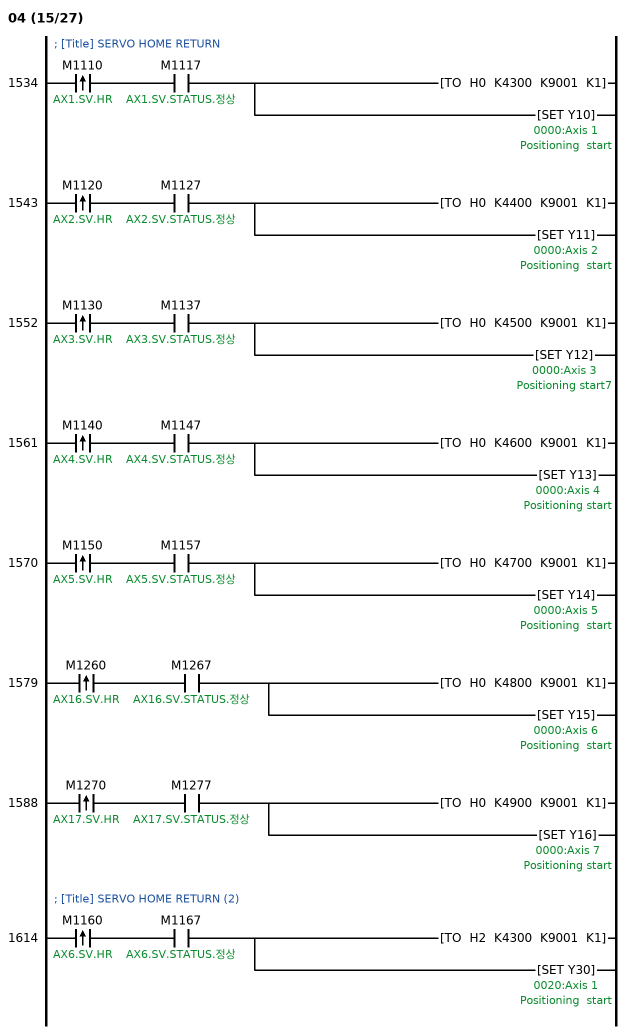
; [Title] SERVO HOME RETURN
1534  LDP     M1110  ; AX1.SV.HR
      AND     M1117  ; AX1.SV.STATUS.정상
      TO      H0 K4300 K9001 K1
      SET     Y10  ; 0000:Axis 1  Positioning  start
1543  LDP     M1120  ; AX2.SV.HR
      AND     M1127  ; AX2.SV.STATUS.정상
      TO      H0 K4400 K9001 K1
      SET     Y11  ; 0000:Axis 2  Positioning  start
1552  LDP     M1130  ; AX3.SV.HR
      AND     M1137  ; AX3.SV.STATUS.정상
      TO      H0 K4500 K9001 K1
      SET     Y12  ; 0000:Axis 3 Positioning start7
1561  LDP     M1140  ; AX4.SV.HR
      AND     M1147  ; AX4.SV.STATUS.정상
      TO      H0 K4600 K9001 K1
      SET     Y13  ; 0000:Axis 4 Positioning start
1570  LDP     M1150  ; AX5.SV.HR
      AND     M1157  ; AX5.SV.STATUS.정상
      TO      H0 K4700 K9001 K1
      SET     Y14  ; 0000:Axis 5  Positioning  start
1579  LDP     M1260  ; AX16.SV.HR
      AND     M1267  ; AX16.SV.STATUS.정상
      TO      H0 K4800 K9001 K1
      SET     Y15  ; 0000:Axis 6  Positioning  start
1588  LDP     M1270  ; AX17.SV.HR
      AND     M1277  ; AX17.SV.STATUS.정상
      TO      H0 K4900 K9001 K1
      SET     Y16  ; 0000:Axis 7 Positioning start
; [Title] SERVO HOME RETURN (2)
1614  LDP     M1160  ; AX6.SV.HR
      AND     M1167  ; AX6.SV.STATUS.정상
      TO      H2 K4300 K9001 K1
      SET     Y30  ; 0020:Axis 1  Positioning  start
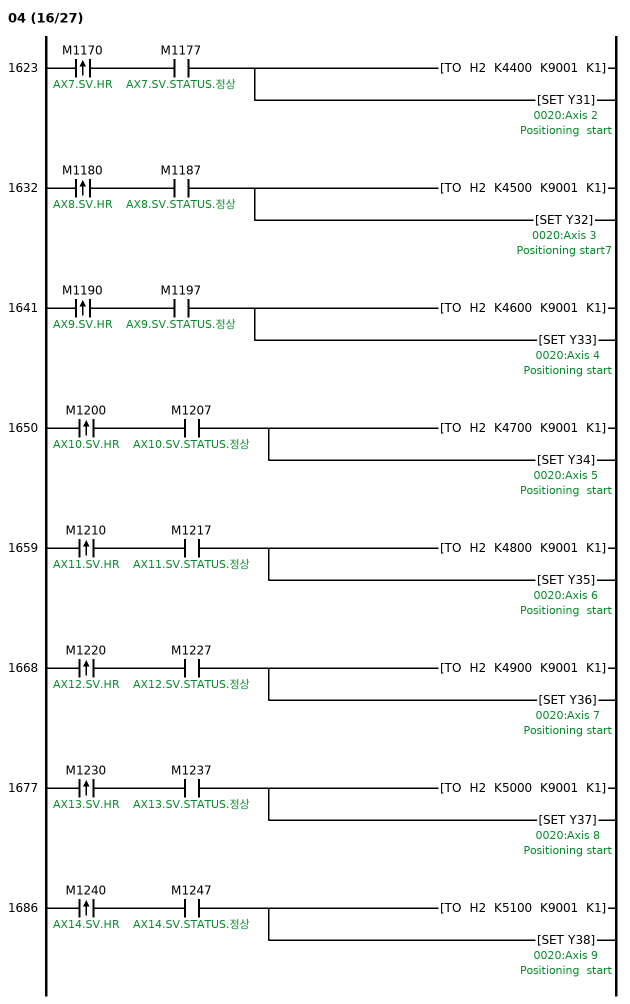
1623  LDP     M1170  ; AX7.SV.HR
      AND     M1177  ; AX7.SV.STATUS.정상
      TO      H2 K4400 K9001 K1
      SET     Y31  ; 0020:Axis 2  Positioning  start
1632  LDP     M1180  ; AX8.SV.HR
      AND     M1187  ; AX8.SV.STATUS.정상
      TO      H2 K4500 K9001 K1
      SET     Y32  ; 0020:Axis 3 Positioning start7
1641  LDP     M1190  ; AX9.SV.HR
      AND     M1197  ; AX9.SV.STATUS.정상
      TO      H2 K4600 K9001 K1
      SET     Y33  ; 0020:Axis 4 Positioning start
1650  LDP     M1200  ; AX10.SV.HR
      AND     M1207  ; AX10.SV.STATUS.정상
      TO      H2 K4700 K9001 K1
      SET     Y34  ; 0020:Axis 5  Positioning  start
1659  LDP     M1210  ; AX11.SV.HR
      AND     M1217  ; AX11.SV.STATUS.정상
      TO      H2 K4800 K9001 K1
      SET     Y35  ; 0020:Axis 6  Positioning  start
1668  LDP     M1220  ; AX12.SV.HR
      AND     M1227  ; AX12.SV.STATUS.정상
      TO      H2 K4900 K9001 K1
      SET     Y36  ; 0020:Axis 7 Positioning start
1677  LDP     M1230  ; AX13.SV.HR
      AND     M1237  ; AX13.SV.STATUS.정상
      TO      H2 K5000 K9001 K1
      SET     Y37  ; 0020:Axis 8 Positioning start
1686  LDP     M1240  ; AX14.SV.HR
      AND     M1247  ; AX14.SV.STATUS.정상
      TO      H2 K5100 K9001 K1
      SET     Y38  ; 0020:Axis 9  Positioning  start
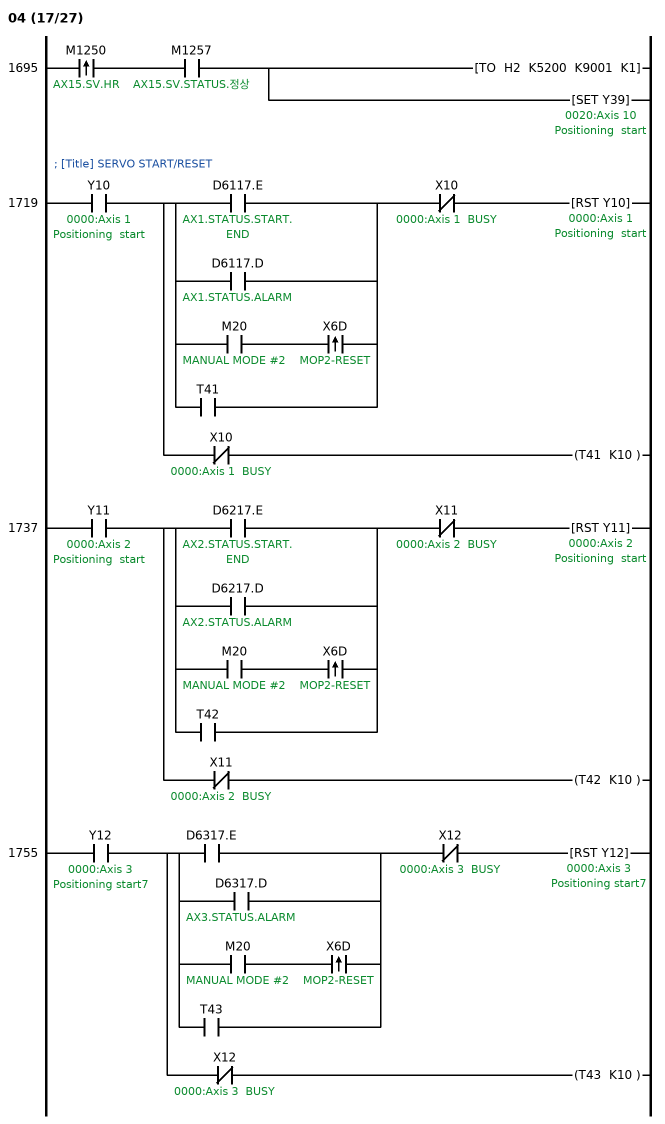
1695  LDP     M1250  ; AX15.SV.HR
      AND     M1257  ; AX15.SV.STATUS.정상
      TO      H2 K5200 K9001 K1
      SET     Y39  ; 0020:Axis 10  Positioning  start
; [Title] SERVO START/RESET
1719  LD      Y10  ; 0000:Axis 1  Positioning  start
      MPS
      LD      D6117.E  ; AX1.STATUS.START.END
      OR      D6117.D  ; AX1.STATUS.ALARM
      LD      M20  ; MANUAL MODE #2
      ANDP    X6D  ; MOP2-RESET
      ORB
      OR      T41
      ANB
      ANI     X10  ; 0000:Axis 1  BUSY
      RST     Y10  ; 0000:Axis 1  Positioning  start
      MPP
      ANI     X10  ; 0000:Axis 1  BUSY
      OUT     T41 K10
1737  LD      Y11  ; 0000:Axis 2  Positioning  start
      MPS
      LD      D6217.E  ; AX2.STATUS.START.END
      OR      D6217.D  ; AX2.STATUS.ALARM
      LD      M20  ; MANUAL MODE #2
      ANDP    X6D  ; MOP2-RESET
      ORB
      OR      T42
      ANB
      ANI     X11  ; 0000:Axis 2  BUSY
      RST     Y11  ; 0000:Axis 2  Positioning  start
      MPP
      ANI     X11  ; 0000:Axis 2  BUSY
      OUT     T42 K10
1755  LD      Y12  ; 0000:Axis 3 Positioning start7
      MPS
      LD      D6317.E
      OR      D6317.D  ; AX3.STATUS.ALARM
      LD      M20  ; MANUAL MODE #2
      ANDP    X6D  ; MOP2-RESET
      ORB
      OR      T43
      ANB
      ANI     X12  ; 0000:Axis 3  BUSY
      RST     Y12  ; 0000:Axis 3 Positioning start7
      MPP
      ANI     X12  ; 0000:Axis 3  BUSY
      OUT     T43 K10
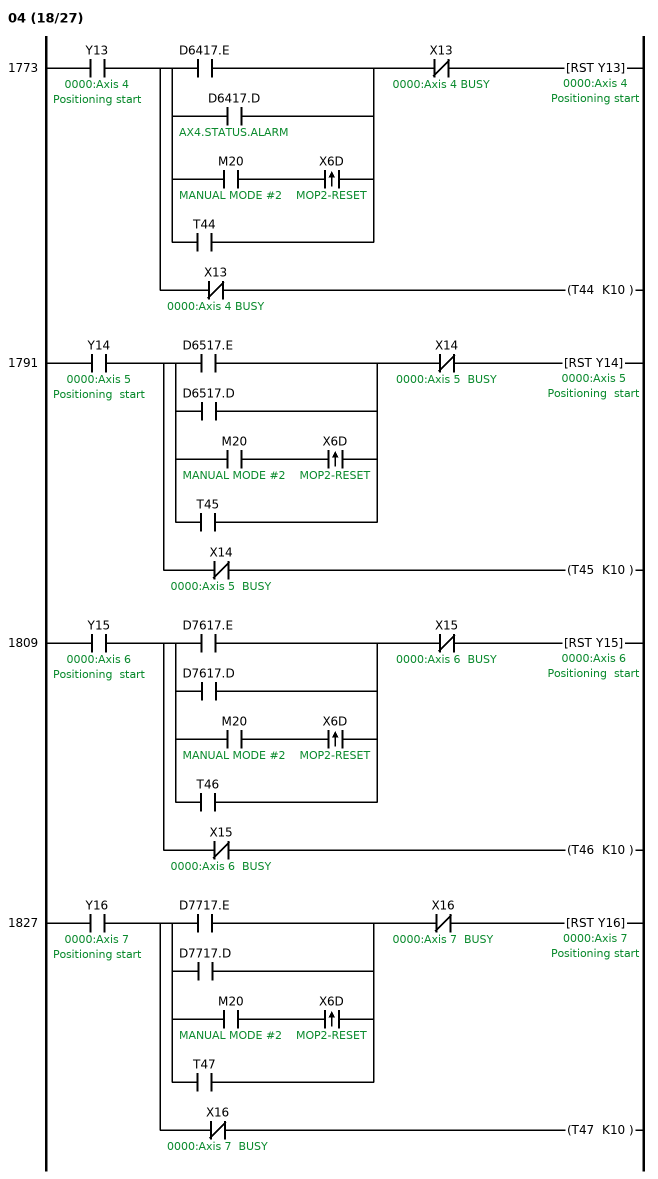
1773  LD      Y13  ; 0000:Axis 4 Positioning start
      MPS
      LD      D6417.E
      OR      D6417.D  ; AX4.STATUS.ALARM
      LD      M20  ; MANUAL MODE #2
      ANDP    X6D  ; MOP2-RESET
      ORB
      OR      T44
      ANB
      ANI     X13  ; 0000:Axis 4 BUSY
      RST     Y13  ; 0000:Axis 4 Positioning start
      MPP
      ANI     X13  ; 0000:Axis 4 BUSY
      OUT     T44 K10
1791  LD      Y14  ; 0000:Axis 5  Positioning  start
      MPS
      LD      D6517.E
      OR      D6517.D
      LD      M20  ; MANUAL MODE #2
      ANDP    X6D  ; MOP2-RESET
      ORB
      OR      T45
      ANB
      ANI     X14  ; 0000:Axis 5  BUSY
      RST     Y14  ; 0000:Axis 5  Positioning  start
      MPP
      ANI     X14  ; 0000:Axis 5  BUSY
      OUT     T45 K10
1809  LD      Y15  ; 0000:Axis 6  Positioning  start
      MPS
      LD      D7617.E
      OR      D7617.D
      LD      M20  ; MANUAL MODE #2
      ANDP    X6D  ; MOP2-RESET
      ORB
      OR      T46
      ANB
      ANI     X15  ; 0000:Axis 6  BUSY
      RST     Y15  ; 0000:Axis 6  Positioning  start
      MPP
      ANI     X15  ; 0000:Axis 6  BUSY
      OUT     T46 K10
1827  LD      Y16  ; 0000:Axis 7 Positioning start
      MPS
      LD      D7717.E
      OR      D7717.D
      LD      M20  ; MANUAL MODE #2
      ANDP    X6D  ; MOP2-RESET
      ORB
      OR      T47
      ANB
      ANI     X16  ; 0000:Axis 7  BUSY
      RST     Y16  ; 0000:Axis 7 Positioning start
      MPP
      ANI     X16  ; 0000:Axis 7  BUSY
      OUT     T47 K10
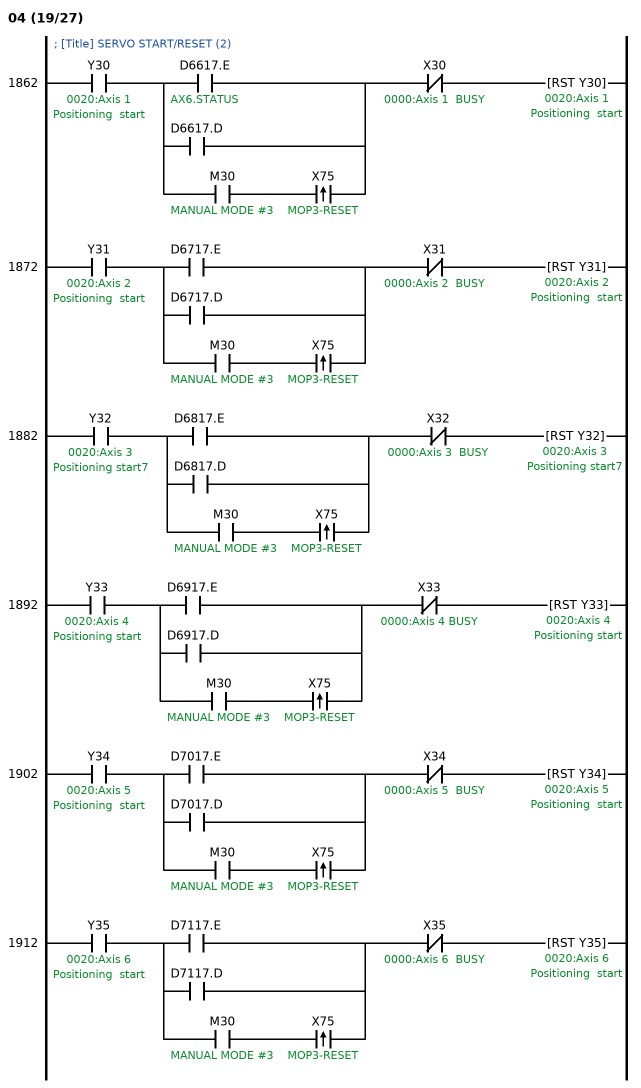
; [Title] SERVO START/RESET (2)
1862  LD      Y30  ; 0020:Axis 1  Positioning  start
      LD      D6617.E  ; AX6.STATUS
      OR      D6617.D
      LD      M30  ; MANUAL MODE #3
      ANDP    X75  ; MOP3-RESET
      ORB
      ANB
      ANI     X30  ; 0000:Axis 1  BUSY
      RST     Y30  ; 0020:Axis 1  Positioning  start
1872  LD      Y31  ; 0020:Axis 2  Positioning  start
      LD      D6717.E
      OR      D6717.D
      LD      M30  ; MANUAL MODE #3
      ANDP    X75  ; MOP3-RESET
      ORB
      ANB
      ANI     X31  ; 0000:Axis 2  BUSY
      RST     Y31  ; 0020:Axis 2  Positioning  start
1882  LD      Y32  ; 0020:Axis 3 Positioning start7
      LD      D6817.E
      OR      D6817.D
      LD      M30  ; MANUAL MODE #3
      ANDP    X75  ; MOP3-RESET
      ORB
      ANB
      ANI     X32  ; 0000:Axis 3  BUSY
      RST     Y32  ; 0020:Axis 3 Positioning start7
1892  LD      Y33  ; 0020:Axis 4 Positioning start
      LD      D6917.E
      OR      D6917.D
      LD      M30  ; MANUAL MODE #3
      ANDP    X75  ; MOP3-RESET
      ORB
      ANB
      ANI     X33  ; 0000:Axis 4 BUSY
      RST     Y33  ; 0020:Axis 4 Positioning start
1902  LD      Y34  ; 0020:Axis 5  Positioning  start
      LD      D7017.E
      OR      D7017.D
      LD      M30  ; MANUAL MODE #3
      ANDP    X75  ; MOP3-RESET
      ORB
      ANB
      ANI     X34  ; 0000:Axis 5  BUSY
      RST     Y34  ; 0020:Axis 5  Positioning  start
1912  LD      Y35  ; 0020:Axis 6  Positioning  start
      LD      D7117.E
      OR      D7117.D
      LD      M30  ; MANUAL MODE #3
      ANDP    X75  ; MOP3-RESET
      ORB
      ANB
      ANI     X35  ; 0000:Axis 6  BUSY
      RST     Y35  ; 0020:Axis 6  Positioning  start
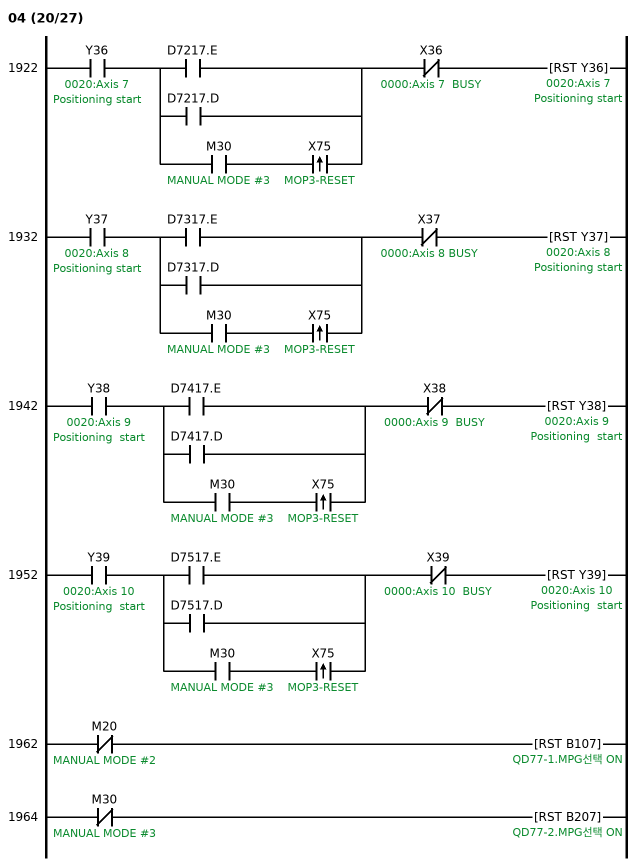
1922  LD      Y36  ; 0020:Axis 7 Positioning start
      LD      D7217.E
      OR      D7217.D
      LD      M30  ; MANUAL MODE #3
      ANDP    X75  ; MOP3-RESET
      ORB
      ANB
      ANI     X36  ; 0000:Axis 7  BUSY
      RST     Y36  ; 0020:Axis 7 Positioning start
1932  LD      Y37  ; 0020:Axis 8 Positioning start
      LD      D7317.E
      OR      D7317.D
      LD      M30  ; MANUAL MODE #3
      ANDP    X75  ; MOP3-RESET
      ORB
      ANB
      ANI     X37  ; 0000:Axis 8 BUSY
      RST     Y37  ; 0020:Axis 8 Positioning start
1942  LD      Y38  ; 0020:Axis 9  Positioning  start
      LD      D7417.E
      OR      D7417.D
      LD      M30  ; MANUAL MODE #3
      ANDP    X75  ; MOP3-RESET
      ORB
      ANB
      ANI     X38  ; 0000:Axis 9  BUSY
      RST     Y38  ; 0020:Axis 9  Positioning  start
1952  LD      Y39  ; 0020:Axis 10  Positioning  start
      LD      D7517.E
      OR      D7517.D
      LD      M30  ; MANUAL MODE #3
      ANDP    X75  ; MOP3-RESET
      ORB
      ANB
      ANI     X39  ; 0000:Axis 10  BUSY
      RST     Y39  ; 0020:Axis 10  Positioning  start
1962  LDI     M20  ; MANUAL MODE #2
      RST     B107  ; QD77-1.MPG선택 ON
1964  LDI     M30  ; MANUAL MODE #3
      RST     B207  ; QD77-2.MPG선택 ON
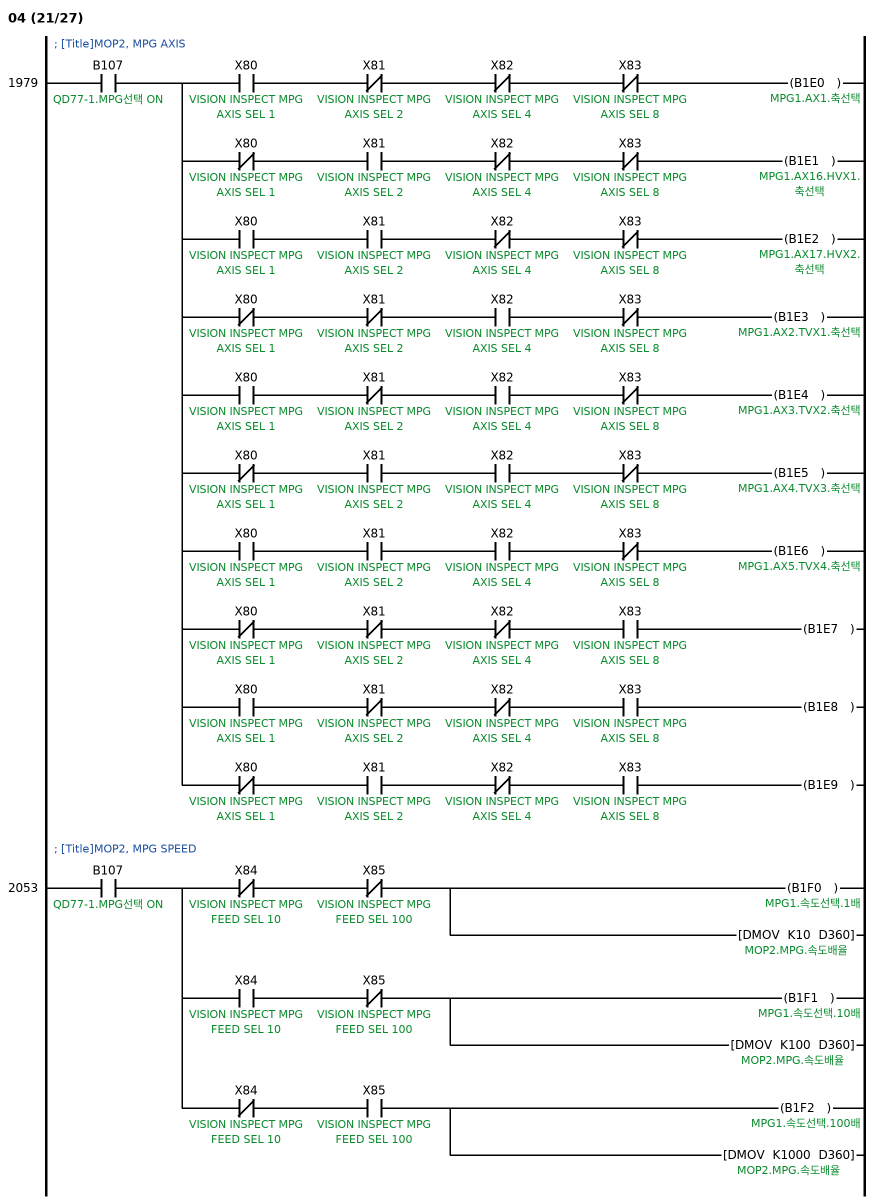
; [Title]MOP2, MPG AXIS
1979  LD      B107  ; QD77-1.MPG선택 ON
      MPS
      AND     X80  ; VISION INSPECT MPG AXIS SEL 1
      ANI     X81  ; VISION INSPECT MPG AXIS SEL 2
      ANI     X82  ; VISION INSPECT MPG AXIS SEL 4
      ANI     X83  ; VISION INSPECT MPG AXIS SEL 8
      OUT     B1E0  ; MPG1.AX1.축선택
      MRD
      ANI     X80  ; VISION INSPECT MPG AXIS SEL 1
      AND     X81  ; VISION INSPECT MPG AXIS SEL 2
      ANI     X82  ; VISION INSPECT MPG AXIS SEL 4
      ANI     X83  ; VISION INSPECT MPG AXIS SEL 8
      OUT     B1E1  ; MPG1.AX16.HVX1.축선택
      MRD
      AND     X80  ; VISION INSPECT MPG AXIS SEL 1
      AND     X81  ; VISION INSPECT MPG AXIS SEL 2
      ANI     X82  ; VISION INSPECT MPG AXIS SEL 4
      ANI     X83  ; VISION INSPECT MPG AXIS SEL 8
      OUT     B1E2  ; MPG1.AX17.HVX2.축선택
      MRD
      ANI     X80  ; VISION INSPECT MPG AXIS SEL 1
      ANI     X81  ; VISION INSPECT MPG AXIS SEL 2
      AND     X82  ; VISION INSPECT MPG AXIS SEL 4
      ANI     X83  ; VISION INSPECT MPG AXIS SEL 8
      OUT     B1E3  ; MPG1.AX2.TVX1.축선택
      MRD
      AND     X80  ; VISION INSPECT MPG AXIS SEL 1
      ANI     X81  ; VISION INSPECT MPG AXIS SEL 2
      AND     X82  ; VISION INSPECT MPG AXIS SEL 4
      ANI     X83  ; VISION INSPECT MPG AXIS SEL 8
      OUT     B1E4  ; MPG1.AX3.TVX2.축선택
      MRD
      ANI     X80  ; VISION INSPECT MPG AXIS SEL 1
      AND     X81  ; VISION INSPECT MPG AXIS SEL 2
      AND     X82  ; VISION INSPECT MPG AXIS SEL 4
      ANI     X83  ; VISION INSPECT MPG AXIS SEL 8
      OUT     B1E5  ; MPG1.AX4.TVX3.축선택
      MRD
      AND     X80  ; VISION INSPECT MPG AXIS SEL 1
      AND     X81  ; VISION INSPECT MPG AXIS SEL 2
      AND     X82  ; VISION INSPECT MPG AXIS SEL 4
      ANI     X83  ; VISION INSPECT MPG AXIS SEL 8
      OUT     B1E6  ; MPG1.AX5.TVX4.축선택
      MRD
      ANI     X80  ; VISION INSPECT MPG AXIS SEL 1
      ANI     X81  ; VISION INSPECT MPG AXIS SEL 2
      ANI     X82  ; VISION INSPECT MPG AXIS SEL 4
      AND     X83  ; VISION INSPECT MPG AXIS SEL 8
      OUT     B1E7
      MRD
      AND     X80  ; VISION INSPECT MPG AXIS SEL 1
      ANI     X81  ; VISION INSPECT MPG AXIS SEL 2
      ANI     X82  ; VISION INSPECT MPG AXIS SEL 4
      AND     X83  ; VISION INSPECT MPG AXIS SEL 8
      OUT     B1E8
      MPP
      ANI     X80  ; VISION INSPECT MPG AXIS SEL 1
      AND     X81  ; VISION INSPECT MPG AXIS SEL 2
      ANI     X82  ; VISION INSPECT MPG AXIS SEL 4
      AND     X83  ; VISION INSPECT MPG AXIS SEL 8
      OUT     B1E9
; [Title]MOP2, MPG SPEED
2053  LD      B107  ; QD77-1.MPG선택 ON
      MPS
      ANI     X84  ; VISION INSPECT MPG FEED SEL 10
      ANI     X85  ; VISION INSPECT MPG FEED SEL 100
      OUT     B1F0  ; MPG1.속도선택.1배
      DMOV    K10 D360  ; MOP2.MPG.속도배율
      MRD
      AND     X84  ; VISION INSPECT MPG FEED SEL 10
      ANI     X85  ; VISION INSPECT MPG FEED SEL 100
      OUT     B1F1  ; MPG1.속도선택.10배
      DMOV    K100 D360
      MPP
      ANI     X84  ; VISION INSPECT MPG FEED SEL 10
      AND     X85  ; VISION INSPECT MPG FEED SEL 100
      OUT     B1F2  ; MPG1.속도선택.100배
      DMOV    K1000 D360
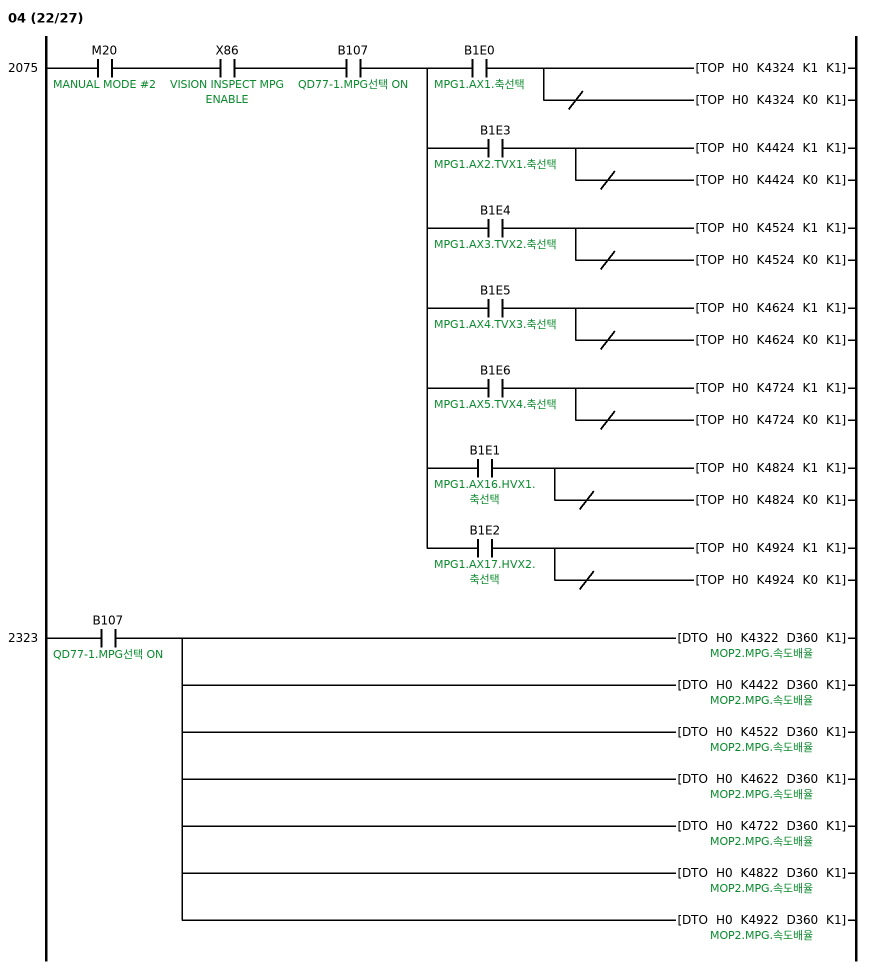
2075  LD      M20  ; MANUAL MODE #2
      AND     X86  ; VISION INSPECT MPG ENABLE
      AND     B107  ; QD77-1.MPG선택 ON
      MPS
      AND     B1E0  ; MPG1.AX1.축선택
      TOP     H0 K4324 K1 K1
        [note] MPG #1 AXIS 허가
      INV
      TOP     H0 K4324 K0 K1
        [note] MPG #1 AXIS 불가
      MRD
      AND     B1E3  ; MPG1.AX2.TVX1.축선택
      TOP     H0 K4424 K1 K1
        [note] MPG #2 AXIS 허가
      INV
      TOP     H0 K4424 K0 K1
        [note] MPG #2 AXIS 불가
      MRD
      AND     B1E4  ; MPG1.AX3.TVX2.축선택
      TOP     H0 K4524 K1 K1
        [note] MPG #3 AXIS 허가
      INV
      TOP     H0 K4524 K0 K1
        [note] MPG #3 AXIS 불가
      MRD
      AND     B1E5  ; MPG1.AX4.TVX3.축선택
      TOP     H0 K4624 K1 K1
        [note] MPG #4 AXIS 허가
      INV
      TOP     H0 K4624 K0 K1
        [note] MPG #4 AXIS 불가
      MRD
      AND     B1E6  ; MPG1.AX5.TVX4.축선택
      TOP     H0 K4724 K1 K1
        [note] MPG #5 AXIS 허가
      INV
      TOP     H0 K4724 K0 K1
        [note] MPG #5 AXIS 불가
      MRD
      AND     B1E1  ; MPG1.AX16.HVX1.축선택
      TOP     H0 K4824 K1 K1
        [note] MPG #6 AXIS 허가
      INV
      TOP     H0 K4824 K0 K1
        [note] MPG #6 AXIS 불가
      MPP
      AND     B1E2  ; MPG1.AX17.HVX2.축선택
      TOP     H0 K4924 K1 K1
        [note] MPG #7 AXIS 허가
      INV
      TOP     H0 K4924 K0 K1
        [note] MPG #7 AXIS 불가
2323  LD      B107  ; QD77-1.MPG선택 ON
      DTO     H0 K4322 D360 K1
      DTO     H0 K4422 D360 K1
      DTO     H0 K4522 D360 K1
      DTO     H0 K4622 D360 K1
      DTO     H0 K4722 D360 K1
      DTO     H0 K4822 D360 K1
      DTO     H0 K4922 D360 K1
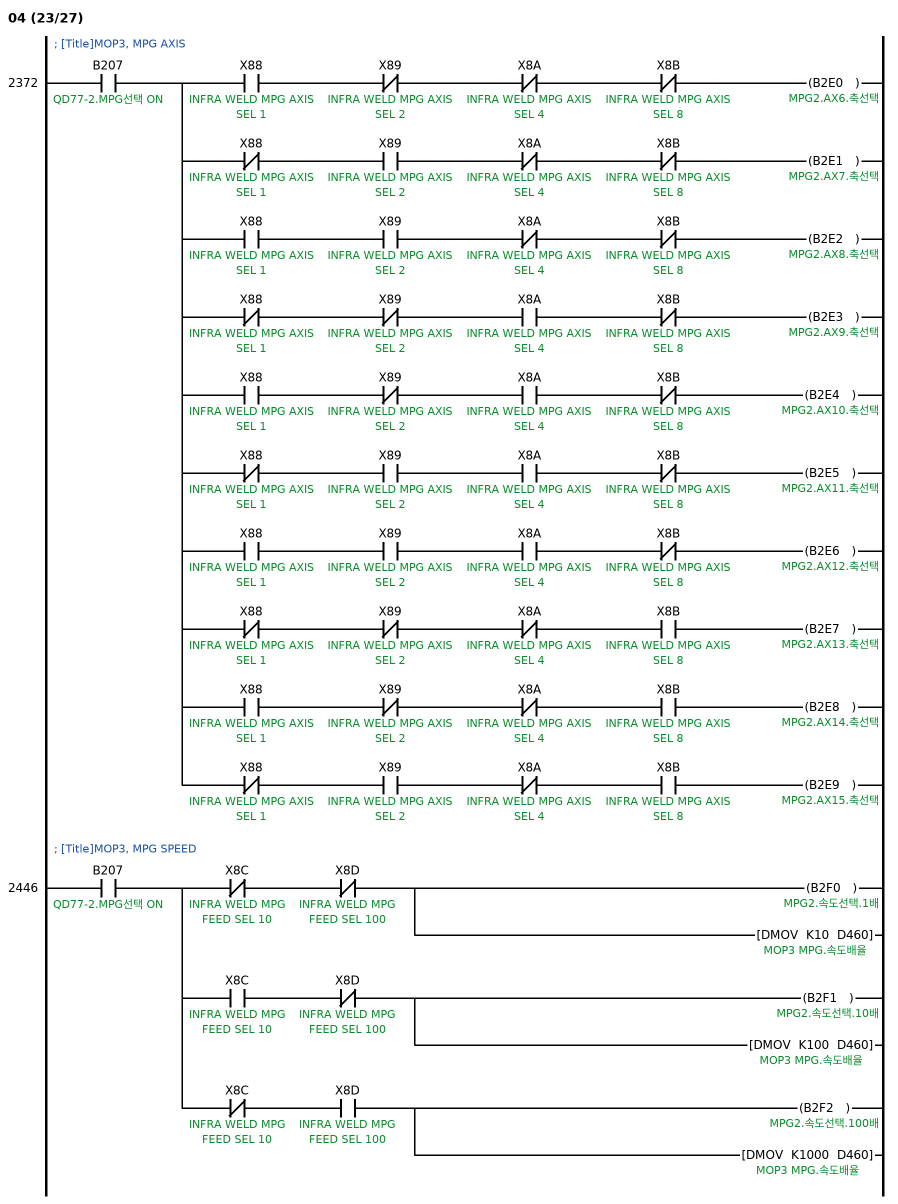
; [Title]MOP3, MPG AXIS
2372  LD      B207  ; QD77-2.MPG선택 ON
      MPS
      AND     X88  ; INFRA WELD MPG AXIS SEL 1
      ANI     X89  ; INFRA WELD MPG AXIS SEL 2
      ANI     X8A  ; INFRA WELD MPG AXIS SEL 4
      ANI     X8B  ; INFRA WELD MPG AXIS SEL 8
      OUT     B2E0  ; MPG2.AX6.축선택
      MRD
      ANI     X88  ; INFRA WELD MPG AXIS SEL 1
      AND     X89  ; INFRA WELD MPG AXIS SEL 2
      ANI     X8A  ; INFRA WELD MPG AXIS SEL 4
      ANI     X8B  ; INFRA WELD MPG AXIS SEL 8
      OUT     B2E1  ; MPG2.AX7.축선택
      MRD
      AND     X88  ; INFRA WELD MPG AXIS SEL 1
      AND     X89  ; INFRA WELD MPG AXIS SEL 2
      ANI     X8A  ; INFRA WELD MPG AXIS SEL 4
      ANI     X8B  ; INFRA WELD MPG AXIS SEL 8
      OUT     B2E2  ; MPG2.AX8.축선택
      MRD
      ANI     X88  ; INFRA WELD MPG AXIS SEL 1
      ANI     X89  ; INFRA WELD MPG AXIS SEL 2
      AND     X8A  ; INFRA WELD MPG AXIS SEL 4
      ANI     X8B  ; INFRA WELD MPG AXIS SEL 8
      OUT     B2E3  ; MPG2.AX9.축선택
      MRD
      AND     X88  ; INFRA WELD MPG AXIS SEL 1
      ANI     X89  ; INFRA WELD MPG AXIS SEL 2
      AND     X8A  ; INFRA WELD MPG AXIS SEL 4
      ANI     X8B  ; INFRA WELD MPG AXIS SEL 8
      OUT     B2E4  ; MPG2.AX10.축선택
      MRD
      ANI     X88  ; INFRA WELD MPG AXIS SEL 1
      AND     X89  ; INFRA WELD MPG AXIS SEL 2
      AND     X8A  ; INFRA WELD MPG AXIS SEL 4
      ANI     X8B  ; INFRA WELD MPG AXIS SEL 8
      OUT     B2E5  ; MPG2.AX11.축선택
      MRD
      AND     X88  ; INFRA WELD MPG AXIS SEL 1
      AND     X89  ; INFRA WELD MPG AXIS SEL 2
      AND     X8A  ; INFRA WELD MPG AXIS SEL 4
      ANI     X8B  ; INFRA WELD MPG AXIS SEL 8
      OUT     B2E6  ; MPG2.AX12.축선택
      MRD
      ANI     X88  ; INFRA WELD MPG AXIS SEL 1
      ANI     X89  ; INFRA WELD MPG AXIS SEL 2
      ANI     X8A  ; INFRA WELD MPG AXIS SEL 4
      AND     X8B  ; INFRA WELD MPG AXIS SEL 8
      OUT     B2E7  ; MPG2.AX13.축선택
      MRD
      AND     X88  ; INFRA WELD MPG AXIS SEL 1
      ANI     X89  ; INFRA WELD MPG AXIS SEL 2
      ANI     X8A  ; INFRA WELD MPG AXIS SEL 4
      AND     X8B  ; INFRA WELD MPG AXIS SEL 8
      OUT     B2E8  ; MPG2.AX14.축선택
      MPP
      ANI     X88  ; INFRA WELD MPG AXIS SEL 1
      AND     X89  ; INFRA WELD MPG AXIS SEL 2
      ANI     X8A  ; INFRA WELD MPG AXIS SEL 4
      AND     X8B  ; INFRA WELD MPG AXIS SEL 8
      OUT     B2E9  ; MPG2.AX15.축선택
; [Title]MOP3, MPG SPEED
2446  LD      B207  ; QD77-2.MPG선택 ON
      MPS
      ANI     X8C  ; INFRA WELD MPG FEED SEL 10
      ANI     X8D  ; INFRA WELD MPG FEED SEL 100
      OUT     B2F0  ; MPG2.속도선택.1배
      DMOV    K10 D460  ; MOP3 MPG.속도배율
      MRD
      AND     X8C  ; INFRA WELD MPG FEED SEL 10
      ANI     X8D  ; INFRA WELD MPG FEED SEL 100
      OUT     B2F1  ; MPG2.속도선택.10배
      DMOV    K100 D460
      MPP
      ANI     X8C  ; INFRA WELD MPG FEED SEL 10
      AND     X8D  ; INFRA WELD MPG FEED SEL 100
      OUT     B2F2  ; MPG2.속도선택.100배
      DMOV    K1000 D460
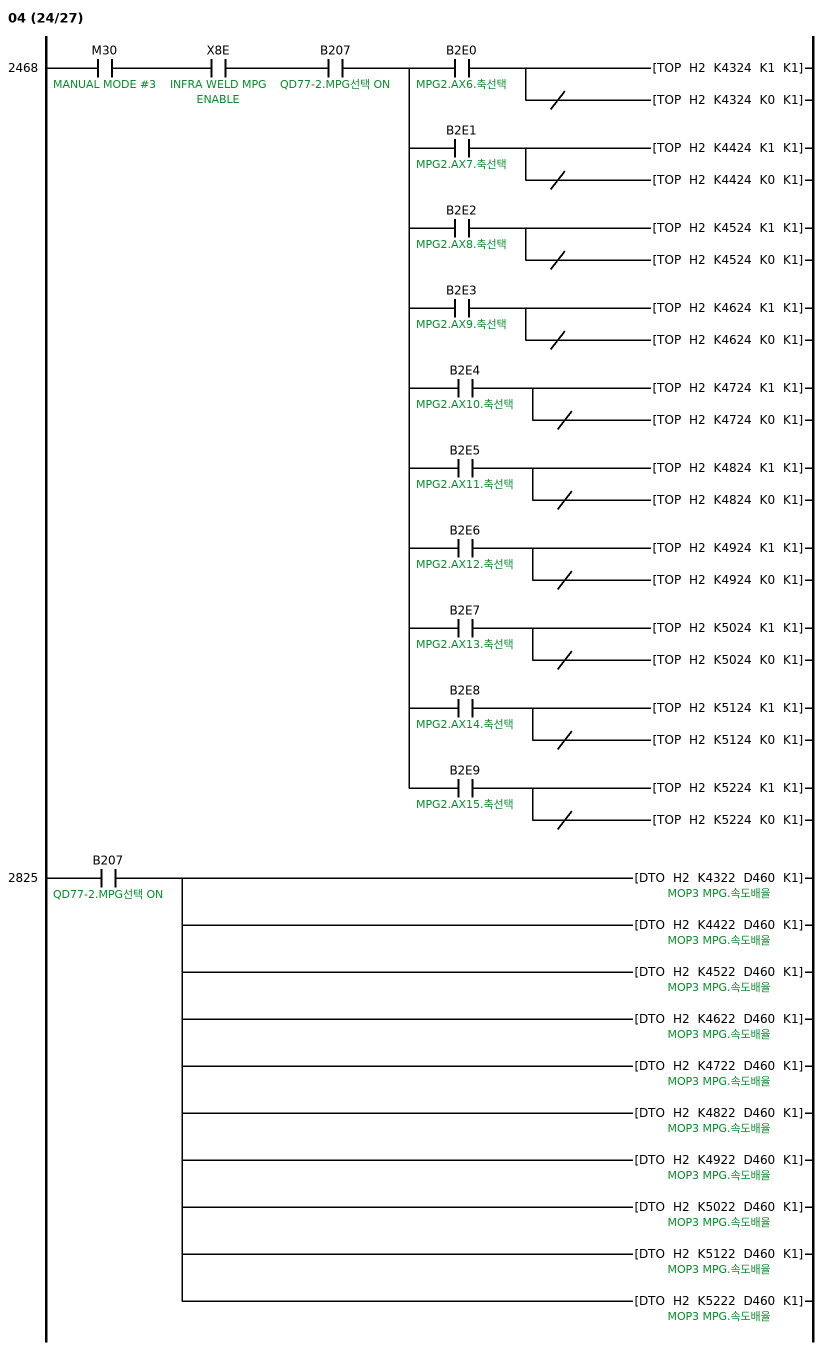
2468  LD      M30  ; MANUAL MODE #3
      AND     X8E  ; INFRA WELD MPG ENABLE
      AND     B207  ; QD77-2.MPG선택 ON
      MPS
      AND     B2E0  ; MPG2.AX6.축선택
      TOP     H2 K4324 K1 K1
        [note] MPG #1 AXIS 허가
      INV
      TOP     H2 K4324 K0 K1
        [note] MPG #1 AXIS 불가
      MRD
      AND     B2E1  ; MPG2.AX7.축선택
      TOP     H2 K4424 K1 K1
        [note] MPG #2 AXIS 허가
      INV
      TOP     H2 K4424 K0 K1
        [note] MPG #2 AXIS 불가
      MRD
      AND     B2E2  ; MPG2.AX8.축선택
      TOP     H2 K4524 K1 K1
        [note] MPG #3 AXIS 허가
      INV
      TOP     H2 K4524 K0 K1
        [note] MPG #3 AXIS 불가
      MRD
      AND     B2E3  ; MPG2.AX9.축선택
      TOP     H2 K4624 K1 K1
        [note] MPG #4 AXIS 허가
      INV
      TOP     H2 K4624 K0 K1
        [note] MPG #4 AXIS 불가
      MRD
      AND     B2E4  ; MPG2.AX10.축선택
      TOP     H2 K4724 K1 K1
        [note] MPG #5 AXIS 허가
      INV
      TOP     H2 K4724 K0 K1
        [note] MPG #5 AXIS 불가
      MRD
      AND     B2E5  ; MPG2.AX11.축선택
      TOP     H2 K4824 K1 K1
        [note] MPG #6 AXIS 허가
      INV
      TOP     H2 K4824 K0 K1
        [note] MPG #5 AXIS 불가
      MRD
      AND     B2E6  ; MPG2.AX12.축선택
      TOP     H2 K4924 K1 K1
        [note] MPG #6 AXIS 허가
      INV
      TOP     H2 K4924 K0 K1
        [note] MPG #5 AXIS 불가
      MRD
      AND     B2E7  ; MPG2.AX13.축선택
      TOP     H2 K5024 K1 K1
        [note] MPG #6 AXIS 허가
      INV
      TOP     H2 K5024 K0 K1
        [note] MPG #5 AXIS 불가
      MRD
      AND     B2E8  ; MPG2.AX14.축선택
      TOP     H2 K5124 K1 K1
        [note] MPG #14 AXIS 허가
      INV
      TOP     H2 K5124 K0 K1
        [note] MPG #14 AXIS 불가
      MPP
      AND     B2E9  ; MPG2.AX15.축선택
      TOP     H2 K5224 K1 K1
        [note] MPG #15 AXIS 허가
      INV
      TOP     H2 K5224 K0 K1
        [note] MPG #15 AXIS 불가
2825  LD      B207  ; QD77-2.MPG선택 ON
      DTO     H2 K4322 D460 K1
      DTO     H2 K4422 D460 K1
      DTO     H2 K4522 D460 K1
      DTO     H2 K4622 D460 K1
      DTO     H2 K4722 D460 K1
      DTO     H2 K4822 D460 K1
      DTO     H2 K4922 D460 K1
      DTO     H2 K5022 D460 K1
      DTO     H2 K5122 D460 K1
      DTO     H2 K5222 D460 K1
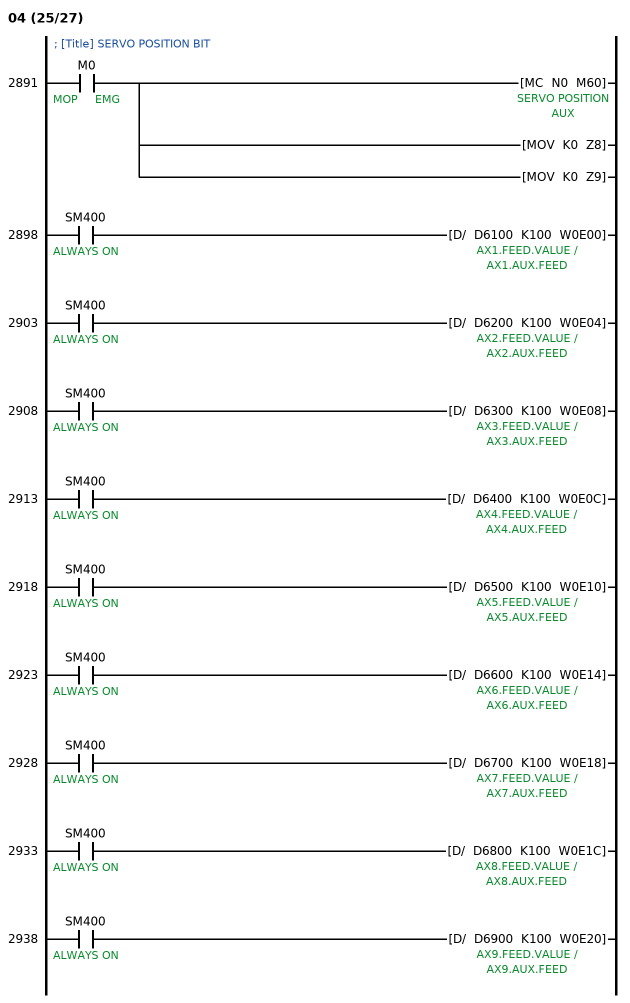
; [Title] SERVO POSITION BIT
2891  LD      M0  ; MOP     EMG
      MC      N0 M60  ; SERVO POSITION AUX
      MOV     K0 Z8
      MOV     K0 Z9
2898  LD      SM400  ; ALWAYS ON
      D/      D6100 K100 W0E00  ; AX1.AUX.FEED
2903  LD      SM400  ; ALWAYS ON
      D/      D6200 K100 W0E04  ; AX2.AUX.FEED
2908  LD      SM400  ; ALWAYS ON
      D/      D6300 K100 W0E08  ; AX3.AUX.FEED
2913  LD      SM400  ; ALWAYS ON
      D/      D6400 K100 W0E0C  ; AX4.AUX.FEED
2918  LD      SM400  ; ALWAYS ON
      D/      D6500 K100 W0E10  ; AX5.AUX.FEED
2923  LD      SM400  ; ALWAYS ON
      D/      D6600 K100 W0E14  ; AX6.AUX.FEED
2928  LD      SM400  ; ALWAYS ON
      D/      D6700 K100 W0E18  ; AX7.AUX.FEED
2933  LD      SM400  ; ALWAYS ON
      D/      D6800 K100 W0E1C  ; AX8.AUX.FEED
2938  LD      SM400  ; ALWAYS ON
      D/      D6900 K100 W0E20  ; AX9.AUX.FEED
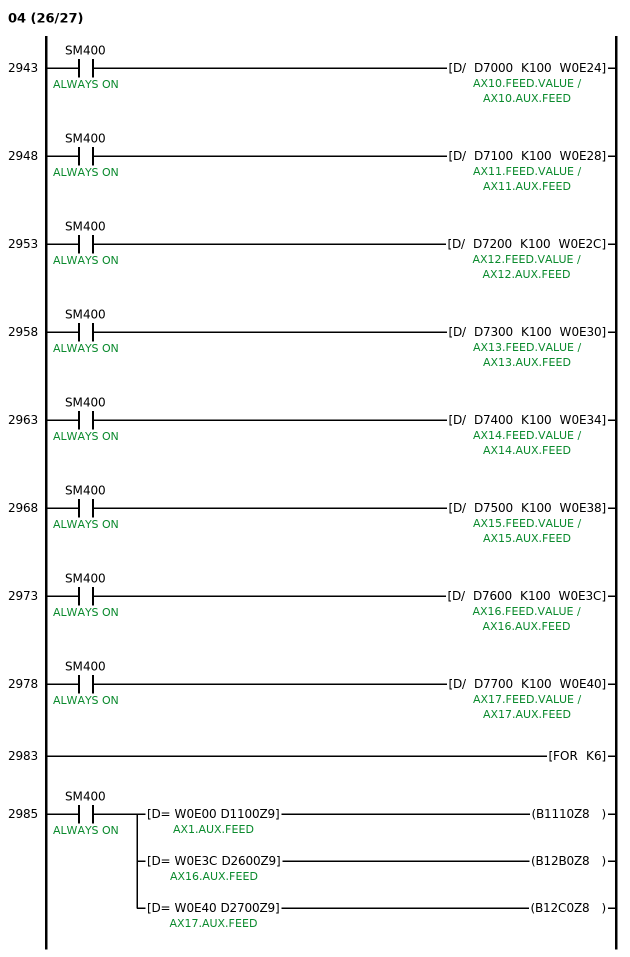
2943  LD      SM400  ; ALWAYS ON
      D/      D7000 K100 W0E24  ; AX10.AUX.FEED
2948  LD      SM400  ; ALWAYS ON
      D/      D7100 K100 W0E28  ; AX11.AUX.FEED
2953  LD      SM400  ; ALWAYS ON
      D/      D7200 K100 W0E2C  ; AX12.AUX.FEED
2958  LD      SM400  ; ALWAYS ON
      D/      D7300 K100 W0E30  ; AX13.AUX.FEED
2963  LD      SM400  ; ALWAYS ON
      D/      D7400 K100 W0E34  ; AX14.AUX.FEED
2968  LD      SM400  ; ALWAYS ON
      D/      D7500 K100 W0E38  ; AX15.AUX.FEED
2973  LD      SM400  ; ALWAYS ON
      D/      D7600 K100 W0E3C  ; AX16.AUX.FEED
2978  LD      SM400  ; ALWAYS ON
      D/      D7700 K100 W0E40  ; AX17.AUX.FEED
2983  FOR     K6
2985  LD      SM400  ; ALWAYS ON
      MPS
      ANDD=   W0E00 D1100Z9  ; AX1.AUX.FEED
      OUT     B1110Z8
      MRD
      ANDD=   W0E3C D2600Z9  ; AX16.AUX.FEED
      OUT     B12B0Z8
      MPP
      ANDD=   W0E40 D2700Z9  ; AX17.AUX.FEED
      OUT     B12C0Z8
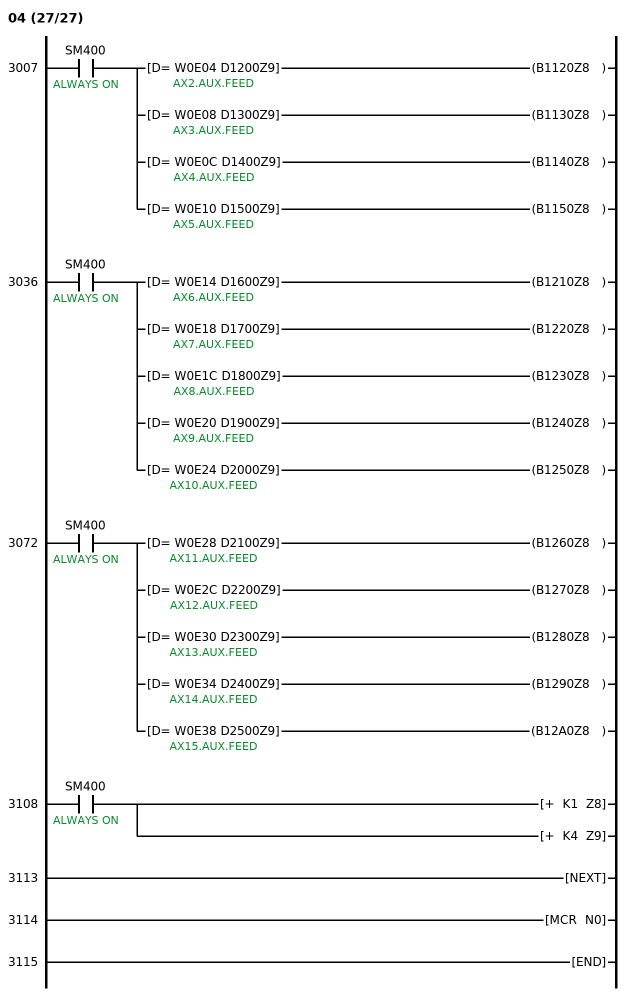
3007  LD      SM400  ; ALWAYS ON
      MPS
      ANDD=   W0E04 D1200Z9  ; AX2.AUX.FEED
      OUT     B1120Z8
      MRD
      ANDD=   W0E08 D1300Z9  ; AX3.AUX.FEED
      OUT     B1130Z8
      MRD
      ANDD=   W0E0C D1400Z9  ; AX4.AUX.FEED
      OUT     B1140Z8
      MPP
      ANDD=   W0E10 D1500Z9  ; AX5.AUX.FEED
      OUT     B1150Z8
3036  LD      SM400  ; ALWAYS ON
      MPS
      ANDD=   W0E14 D1600Z9  ; AX6.AUX.FEED
      OUT     B1210Z8
      MRD
      ANDD=   W0E18 D1700Z9  ; AX7.AUX.FEED
      OUT     B1220Z8
      MRD
      ANDD=   W0E1C D1800Z9  ; AX8.AUX.FEED
      OUT     B1230Z8
      MRD
      ANDD=   W0E20 D1900Z9  ; AX9.AUX.FEED
      OUT     B1240Z8
      MPP
      ANDD=   W0E24 D2000Z9  ; AX10.AUX.FEED
      OUT     B1250Z8
3072  LD      SM400  ; ALWAYS ON
      MPS
      ANDD=   W0E28 D2100Z9  ; AX11.AUX.FEED
      OUT     B1260Z8
      MRD
      ANDD=   W0E2C D2200Z9  ; AX12.AUX.FEED
      OUT     B1270Z8
      MRD
      ANDD=   W0E30 D2300Z9  ; AX13.AUX.FEED
      OUT     B1280Z8
      MRD
      ANDD=   W0E34 D2400Z9  ; AX14.AUX.FEED
      OUT     B1290Z8
      MPP
      ANDD=   W0E38 D2500Z9  ; AX15.AUX.FEED
      OUT     B12A0Z8
3108  LD      SM400  ; ALWAYS ON
      +       K1 Z8
      +       K4 Z9
3113  NEXT
3114  MCR     N0
3115  END
END_PROGRAM

PROGRAM 01  // MAIN
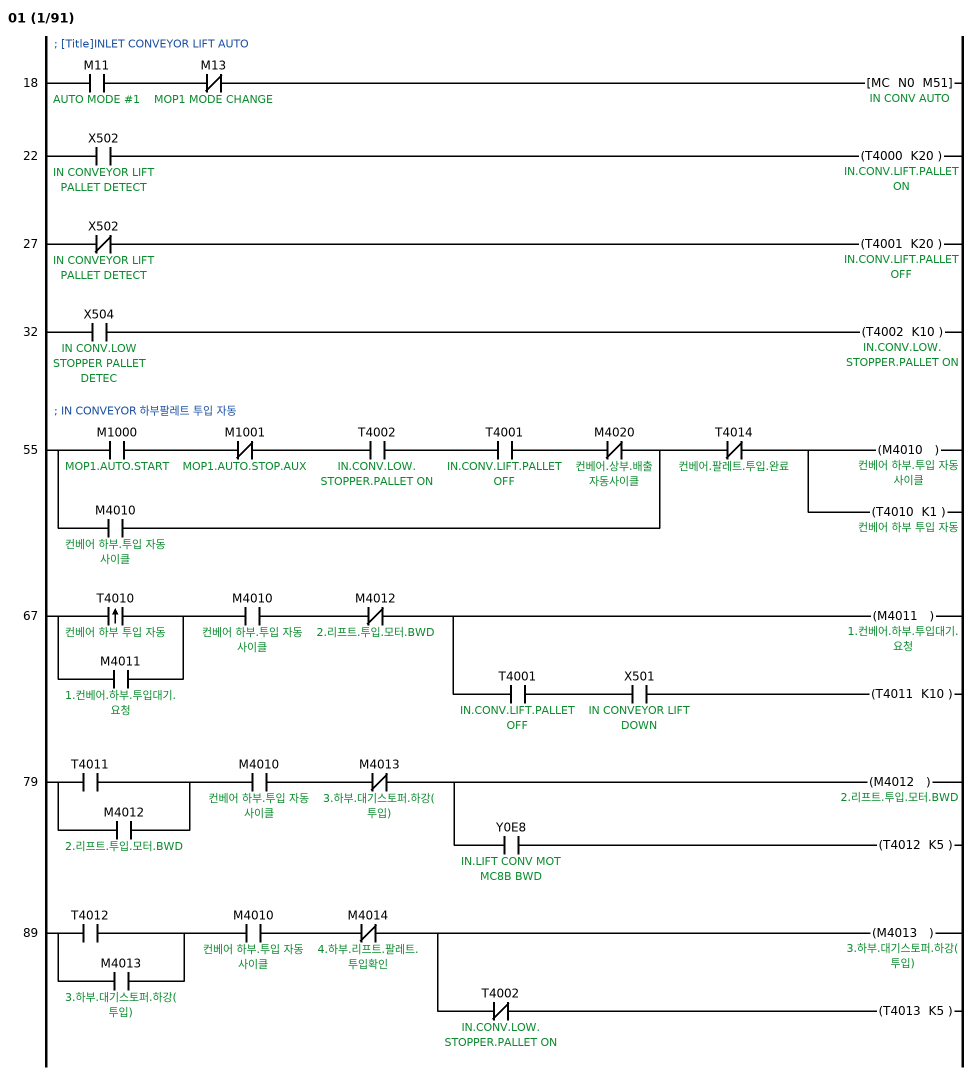
; [Title]INLET CONVEYOR LIFT AUTO
18    LD      M11  ; AUTO MODE #1
      ANI     M13  ; MOP1 MODE CHANGE
      MC      N0 M51  ; IN CONV AUTO
22    LD      X502  ; IN CONVEYOR LIFT PALLET DETECT
      OUT     T4000 K20  ; IN.CONV.LIFT.PALLET ON
27    LDI     X502  ; IN CONVEYOR LIFT PALLET DETECT
      OUT     T4001 K20  ; IN.CONV.LIFT.PALLET OFF
32    LD      X504  ; IN CONV.LOW STOPPER PALLET DETEC
      OUT     T4002 K10  ; IN.CONV.LOW.STOPPER.PALLET ON
; IN CONVEYOR 하부팔레트 투입 자동
55    LD      M1000  ; MOP1.AUTO.START
      ANI     M1001  ; MOP1.AUTO.STOP.AUX
      AND     T4002  ; IN.CONV.LOW.STOPPER.PALLET ON
      AND     T4001  ; IN.CONV.LIFT.PALLET OFF
      ANI     M4020  ; 컨베어.상부.배출 자동사이클
      OR      M4010  ; 컨베어 하부.투입 자동 사이클
      ANI     T4014  ; 컨베어.팔레트.투입.완료
      OUT     M4010  ; 컨베어 하부.투입 자동 사이클
      OUT     T4010 K1  ; 컨베어 하부 투입 자동
67    LDP     T4010  ; 컨베어 하부 투입 자동
      OR      M4011  ; 1.컨베어.하부.투입대기.요청
      AND     M4010  ; 컨베어 하부.투입 자동 사이클
      ANI     M4012  ; 2.리프트.투입.모터.BWD
      OUT     M4011  ; 1.컨베어.하부.투입대기.요청
      AND     T4001  ; IN.CONV.LIFT.PALLET OFF
      AND     X501  ; IN CONVEYOR LIFT DOWN
      OUT     T4011 K10
79    LD      T4011
      OR      M4012  ; 2.리프트.투입.모터.BWD
      AND     M4010  ; 컨베어 하부.투입 자동 사이클
      ANI     M4013  ; 3.하부.대기스토퍼.하강(투입)
      OUT     M4012  ; 2.리프트.투입.모터.BWD
      AND     Y0E8  ; IN.LIFT CONV MOT MC8B BWD
      OUT     T4012 K5
89    LD      T4012
      OR      M4013  ; 3.하부.대기스토퍼.하강(투입)
      AND     M4010  ; 컨베어 하부.투입 자동 사이클
      ANI     M4014  ; 4.하부.리프트.팔레트.투입확인
      OUT     M4013  ; 3.하부.대기스토퍼.하강(투입)
      ANI     T4002  ; IN.CONV.LOW.STOPPER.PALLET ON
      OUT     T4013 K5
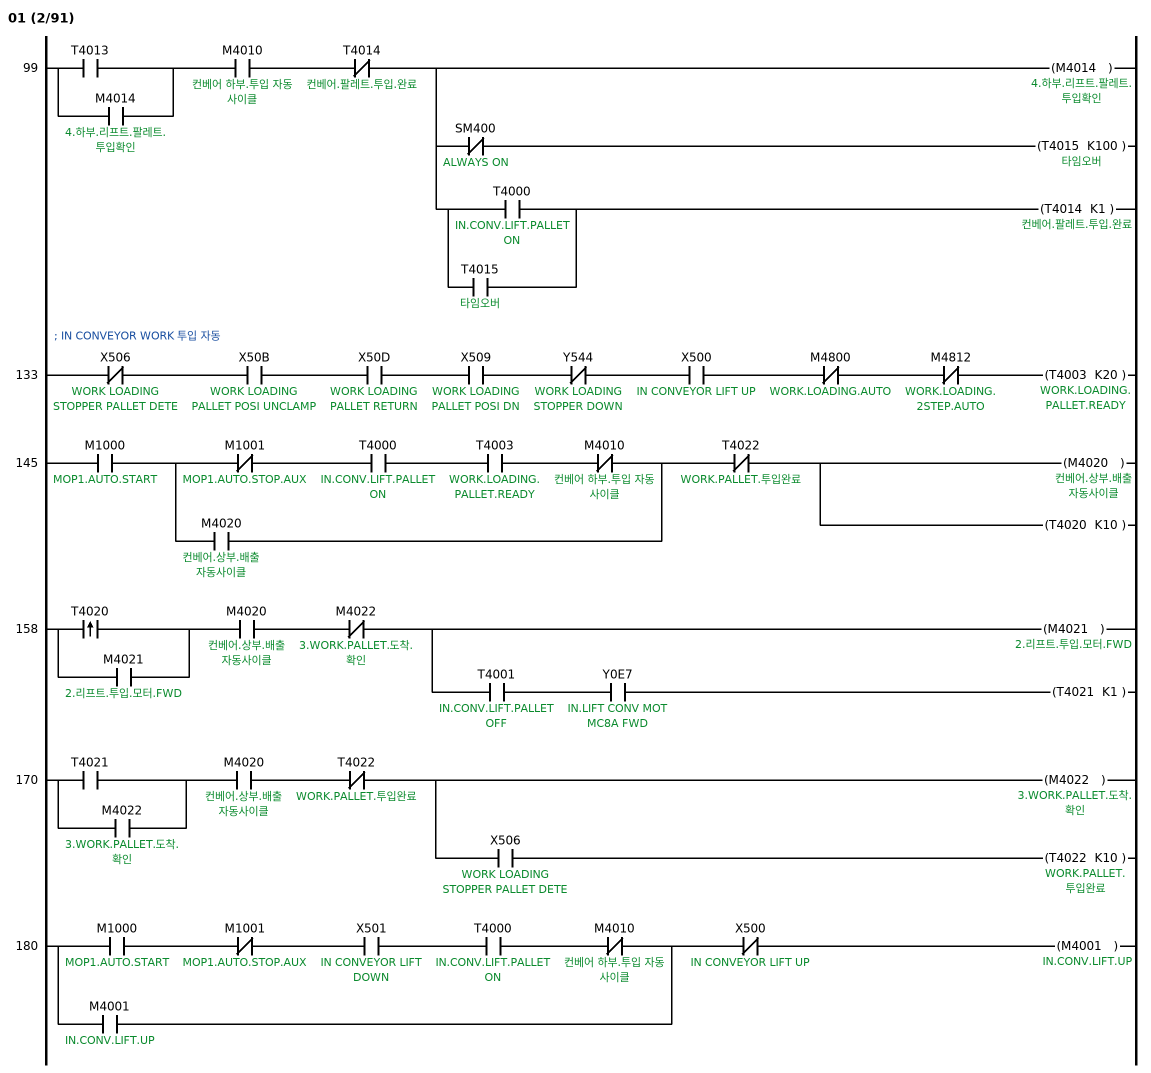
99    LD      T4013
      OR      M4014  ; 4.하부.리프트.팔레트.투입확인
      AND     M4010  ; 컨베어 하부.투입 자동 사이클
      ANI     T4014  ; 컨베어.팔레트.투입.완료
      OUT     M4014  ; 4.하부.리프트.팔레트.투입확인
      MPS
      ANI     SM400  ; ALWAYS ON
      OUT     T4015 K100  ; 타임오버
      MPP
      LD      T4000  ; IN.CONV.LIFT.PALLET ON
      OR      T4015  ; 타임오버
      ANB
      OUT     T4014 K1  ; 컨베어.팔레트.투입.완료
; IN CONVEYOR WORK 투입 자동
133   LDI     X506  ; WORK LOADING STOPPER PALLET DETE
      AND     X50B  ; WORK LOADING PALLET POSI UNCLAMP
      AND     X50D  ; WORK LOADING PALLET RETURN
      AND     X509  ; WORK LOADING PALLET POSI DN
      ANI     Y544  ; WORK LOADING STOPPER DOWN
      AND     X500  ; IN CONVEYOR LIFT UP
      ANI     M4800  ; WORK.LOADING.AUTO
      ANI     M4812  ; WORK.LOADING.2STEP.AUTO
      OUT     T4003 K20  ; WORK.LOADING.PALLET.READY
145   LD      M1000  ; MOP1.AUTO.START
      LDI     M1001  ; MOP1.AUTO.STOP.AUX
      AND     T4000  ; IN.CONV.LIFT.PALLET ON
      AND     T4003  ; WORK.LOADING.PALLET.READY
      ANI     M4010  ; 컨베어 하부.투입 자동 사이클
      OR      M4020  ; 컨베어.상부.배출 자동사이클
      ANB
      ANI     T4022  ; WORK.PALLET.투입완료
      OUT     M4020  ; 컨베어.상부.배출 자동사이클
      OUT     T4020 K10
158   LDP     T4020
      OR      M4021  ; 2.리프트.투입.모터.FWD
      AND     M4020  ; 컨베어.상부.배출 자동사이클
      ANI     M4022  ; 3.WORK.PALLET.도착.확인
      OUT     M4021  ; 2.리프트.투입.모터.FWD
      AND     T4001  ; IN.CONV.LIFT.PALLET OFF
      AND     Y0E7  ; IN.LIFT CONV MOT MC8A FWD
      OUT     T4021 K1
170   LD      T4021
      OR      M4022  ; 3.WORK.PALLET.도착.확인
      AND     M4020  ; 컨베어.상부.배출 자동사이클
      ANI     T4022  ; WORK.PALLET.투입완료
      OUT     M4022  ; 3.WORK.PALLET.도착.확인
      AND     X506  ; WORK LOADING STOPPER PALLET DETE
      OUT     T4022 K10  ; WORK.PALLET.투입완료
180   LD      M1000  ; MOP1.AUTO.START
      ANI     M1001  ; MOP1.AUTO.STOP.AUX
      AND     X501  ; IN CONVEYOR LIFT DOWN
      AND     T4000  ; IN.CONV.LIFT.PALLET ON
      ANI     M4010  ; 컨베어 하부.투입 자동 사이클
      OR      M4001  ; IN.CONV.LIFT.UP
      ANI     X500  ; IN CONVEYOR LIFT UP
      OUT     M4001  ; IN.CONV.LIFT.UP
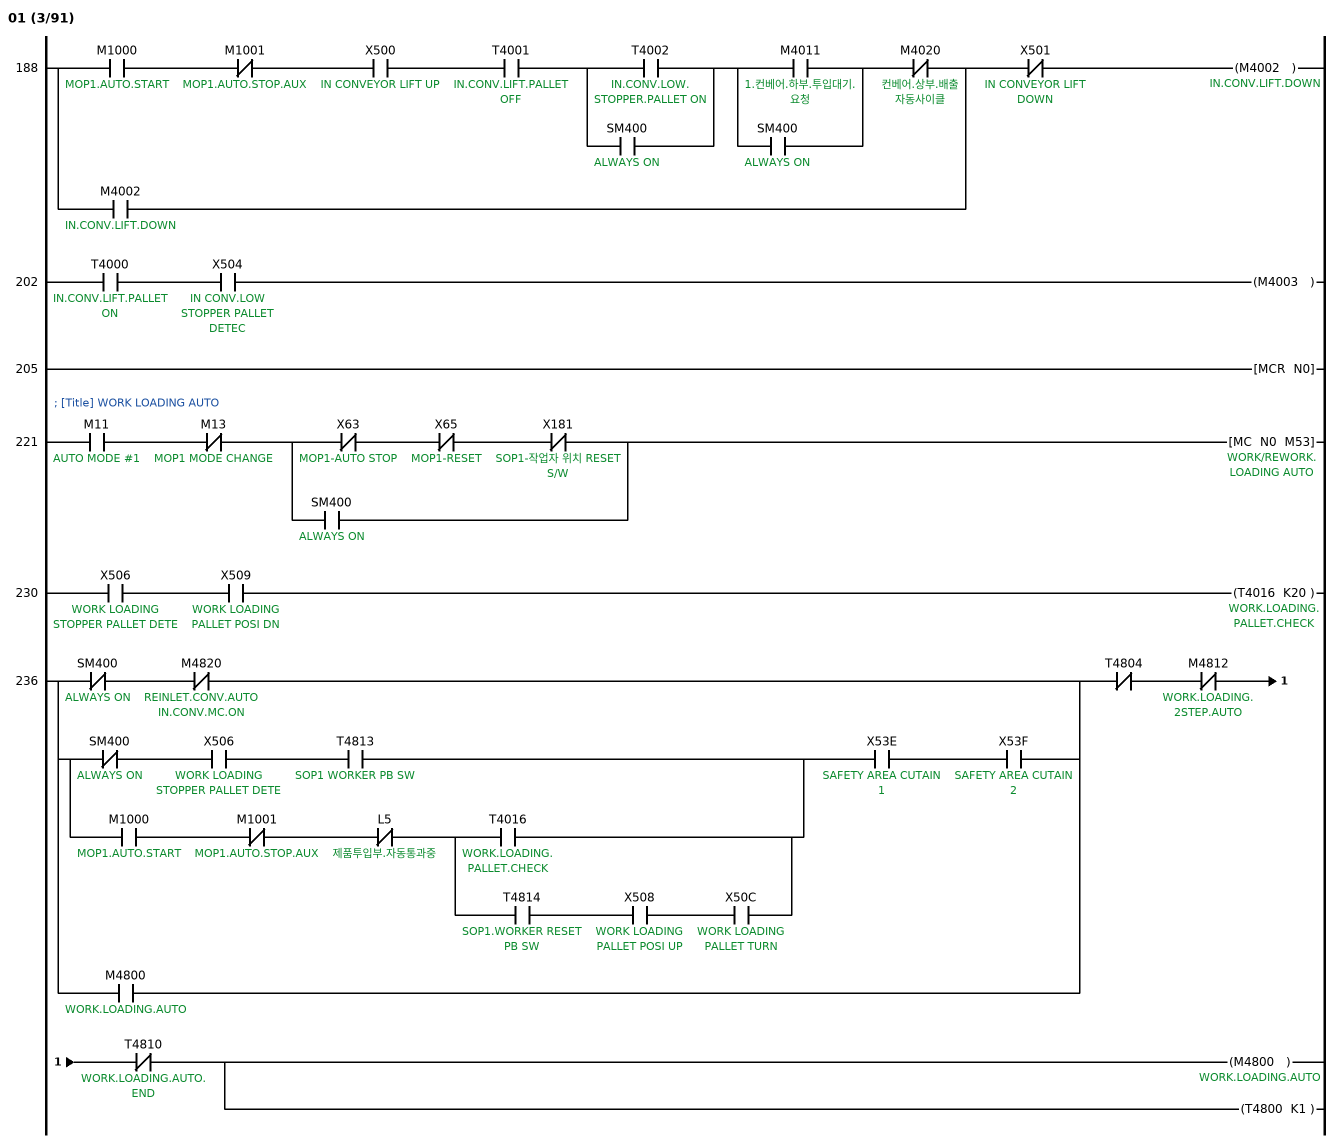
188   LD      M1000  ; MOP1.AUTO.START
      ANI     M1001  ; MOP1.AUTO.STOP.AUX
      AND     X500  ; IN CONVEYOR LIFT UP
      AND     T4001  ; IN.CONV.LIFT.PALLET OFF
      LD      T4002  ; IN.CONV.LOW.STOPPER.PALLET ON
      OR      SM400  ; ALWAYS ON
      ANB
      LD      M4011  ; 1.컨베어.하부.투입대기.요청
      OR      SM400  ; ALWAYS ON
      ANB
      ANI     M4020  ; 컨베어.상부.배출 자동사이클
      OR      M4002  ; IN.CONV.LIFT.DOWN
      ANI     X501  ; IN CONVEYOR LIFT DOWN
      OUT     M4002  ; IN.CONV.LIFT.DOWN
202   LD      T4000  ; IN.CONV.LIFT.PALLET ON
      AND     X504  ; IN CONV.LOW STOPPER PALLET DETEC
      OUT     M4003
205   MCR     N0
; [Title] WORK LOADING AUTO
221   LD      M11  ; AUTO MODE #1
      ANI     M13  ; MOP1 MODE CHANGE
      LDI     X63  ; MOP1-AUTO STOP
      ANI     X65  ; MOP1-RESET
      ANI     X181  ; SOP1-작업자 위치 RESET S/W
      OR      SM400  ; ALWAYS ON
      ANB
      MC      N0 M53  ; WORK/REWORK.LOADING AUTO
230   LD      X506  ; WORK LOADING STOPPER PALLET DETE
      AND     X509  ; WORK LOADING PALLET POSI DN
      OUT     T4016 K20  ; WORK.LOADING.PALLET.CHECK
236   LDI     SM400  ; ALWAYS ON
      ANI     M4820  ; REINLET.CONV.AUTO IN.CONV.MC.ON
      LDI     SM400  ; ALWAYS ON
      AND     X506  ; WORK LOADING STOPPER PALLET DETE
      AND     T4813  ; SOP1 WORKER PB SW
      LD      M1000  ; MOP1.AUTO.START
      ANI     M1001  ; MOP1.AUTO.STOP.AUX
      ANI     L5  ; 제품투입부.자동통과중
      LD      T4016  ; WORK.LOADING.PALLET.CHECK
      LD      T4814  ; SOP1.WORKER RESET PB SW
      AND     X508  ; WORK LOADING PALLET POSI UP
      AND     X50C  ; WORK LOADING PALLET TURN
      ORB
      ANB
      ORB
      AND     X53E  ; SAFETY AREA CUTAIN 1
      AND     X53F  ; SAFETY AREA CUTAIN 2
      ORB
      OR      M4800  ; WORK.LOADING.AUTO
      ANI     T4804
      ANI     M4812  ; WORK.LOADING.2STEP.AUTO
      ANI     T4810  ; WORK.LOADING.AUTO.END
      OUT     M4800  ; WORK.LOADING.AUTO
      OUT     T4800 K1
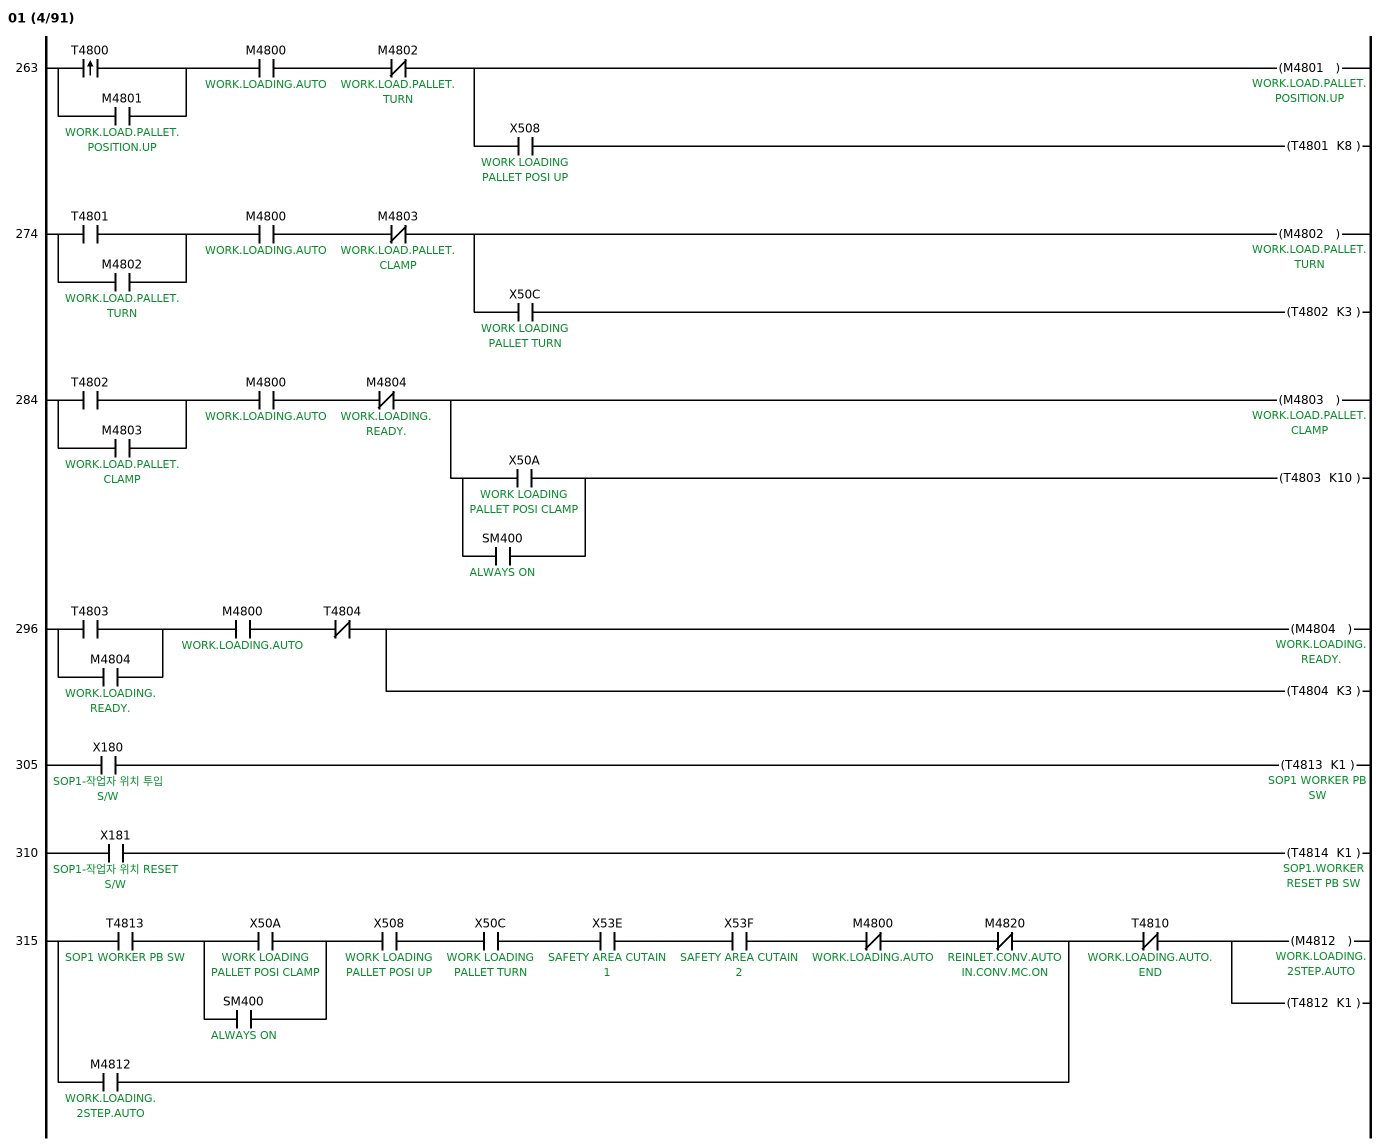
263   LDP     T4800
      OR      M4801  ; WORK.LOAD.PALLET.POSITION.UP
      AND     M4800  ; WORK.LOADING.AUTO
      ANI     M4802  ; WORK.LOAD.PALLET.TURN
      OUT     M4801  ; WORK.LOAD.PALLET.POSITION.UP
      AND     X508  ; WORK LOADING PALLET POSI UP
      OUT     T4801 K8
274   LD      T4801
      OR      M4802  ; WORK.LOAD.PALLET.TURN
      AND     M4800  ; WORK.LOADING.AUTO
      ANI     M4803  ; WORK.LOAD.PALLET.CLAMP
      OUT     M4802  ; WORK.LOAD.PALLET.TURN
      AND     X50C  ; WORK LOADING PALLET TURN
      OUT     T4802 K3
284   LD      T4802
      OR      M4803  ; WORK.LOAD.PALLET.CLAMP
      AND     M4800  ; WORK.LOADING.AUTO
      ANI     M4804  ; WORK.LOADING.READY.
      OUT     M4803  ; WORK.LOAD.PALLET.CLAMP
      LD      X50A  ; WORK LOADING PALLET POSI CLAMP
      OR      SM400  ; ALWAYS ON
      ANB
      OUT     T4803 K10
296   LD      T4803
      OR      M4804  ; WORK.LOADING.READY.
      AND     M4800  ; WORK.LOADING.AUTO
      ANI     T4804
      OUT     M4804  ; WORK.LOADING.READY.
      OUT     T4804 K3
305   LD      X180  ; SOP1-작업자 위치 투입 S/W
      OUT     T4813 K1  ; SOP1 WORKER PB SW
310   LD      X181  ; SOP1-작업자 위치 RESET S/W
      OUT     T4814 K1  ; SOP1.WORKER RESET PB SW
315   LD      T4813  ; SOP1 WORKER PB SW
      LD      X50A  ; WORK LOADING PALLET POSI CLAMP
      OR      SM400  ; ALWAYS ON
      ANB
      AND     X508  ; WORK LOADING PALLET POSI UP
      AND     X50C  ; WORK LOADING PALLET TURN
      AND     X53E  ; SAFETY AREA CUTAIN 1
      AND     X53F  ; SAFETY AREA CUTAIN 2
      ANI     M4800  ; WORK.LOADING.AUTO
      ANI     M4820  ; REINLET.CONV.AUTO IN.CONV.MC.ON
      OR      M4812  ; WORK.LOADING.2STEP.AUTO
      ANI     T4810  ; WORK.LOADING.AUTO.END
      OUT     M4812  ; WORK.LOADING.2STEP.AUTO
      OUT     T4812 K1
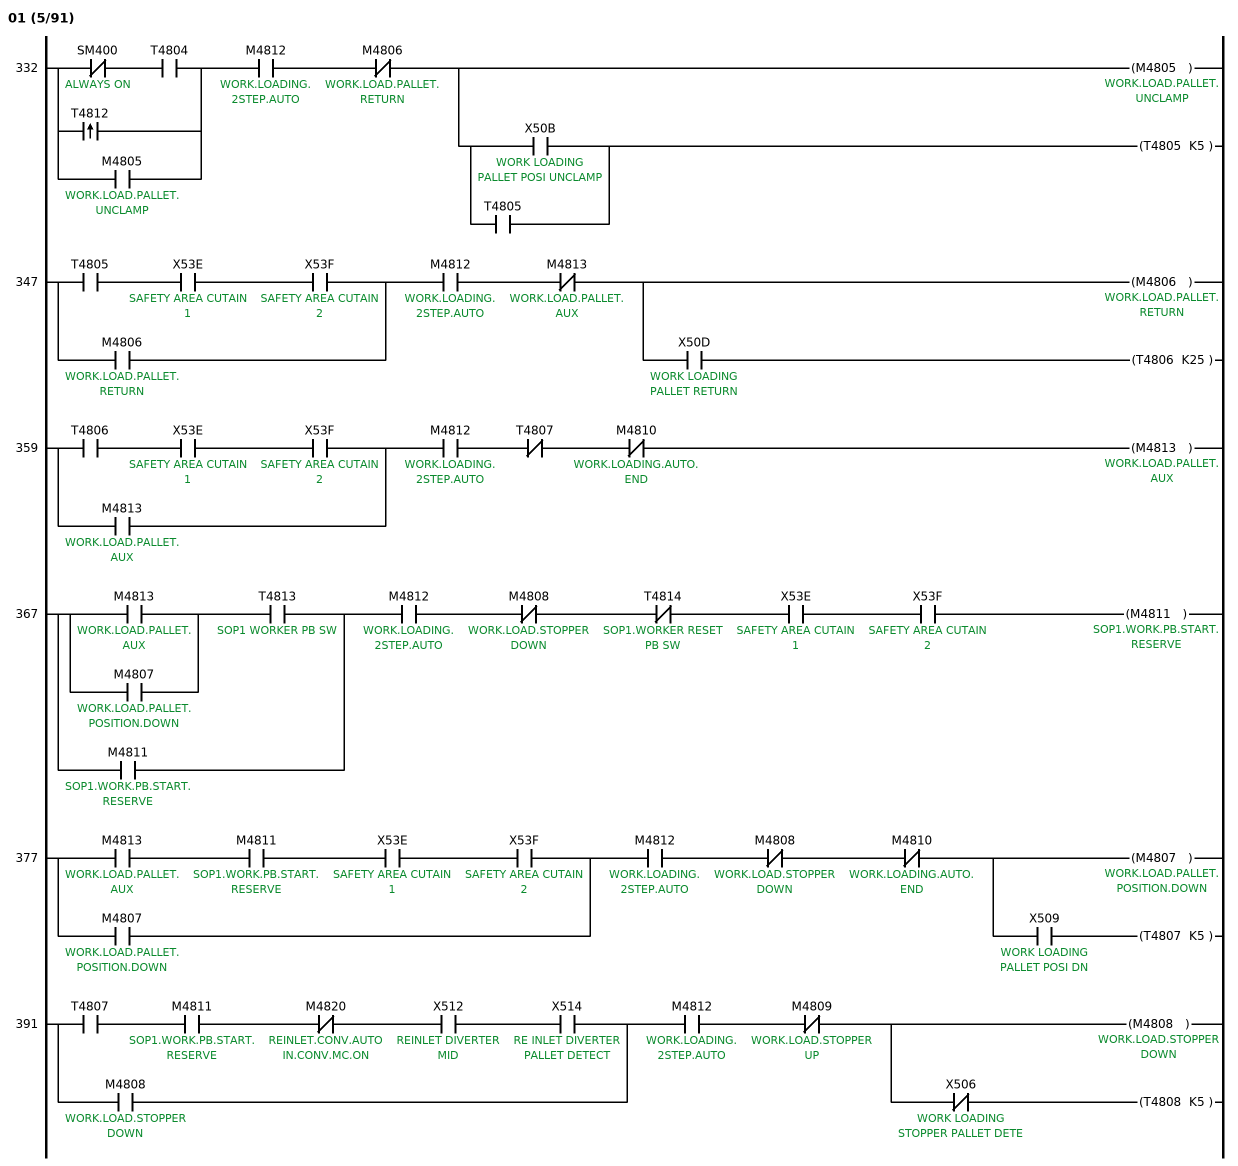
332   LDI     SM400  ; ALWAYS ON
      AND     T4804
      ORP     T4812
      OR      M4805  ; WORK.LOAD.PALLET.UNCLAMP
      AND     M4812  ; WORK.LOADING.2STEP.AUTO
      ANI     M4806  ; WORK.LOAD.PALLET.RETURN
      OUT     M4805  ; WORK.LOAD.PALLET.UNCLAMP
      LD      X50B  ; WORK LOADING PALLET POSI UNCLAMP
      OR      T4805
      ANB
      OUT     T4805 K5
347   LD      T4805
      AND     X53E  ; SAFETY AREA CUTAIN 1
      AND     X53F  ; SAFETY AREA CUTAIN 2
      OR      M4806  ; WORK.LOAD.PALLET.RETURN
      AND     M4812  ; WORK.LOADING.2STEP.AUTO
      ANI     M4813  ; WORK.LOAD.PALLET.AUX
      OUT     M4806  ; WORK.LOAD.PALLET.RETURN
      AND     X50D  ; WORK LOADING PALLET RETURN
      OUT     T4806 K25
359   LD      T4806
      AND     X53E  ; SAFETY AREA CUTAIN 1
      AND     X53F  ; SAFETY AREA CUTAIN 2
      OR      M4813  ; WORK.LOAD.PALLET.AUX
      AND     M4812  ; WORK.LOADING.2STEP.AUTO
      ANI     T4807
      ANI     M4810  ; WORK.LOADING.AUTO.END
      OUT     M4813  ; WORK.LOAD.PALLET.AUX
367   LD      M4813  ; WORK.LOAD.PALLET.AUX
      OR      M4807  ; WORK.LOAD.PALLET.POSITION.DOWN
      AND     T4813  ; SOP1 WORKER PB SW
      OR      M4811  ; SOP1.WORK.PB.START.RESERVE
      AND     M4812  ; WORK.LOADING.2STEP.AUTO
      ANI     M4808  ; WORK.LOAD.STOPPER DOWN
      ANI     T4814  ; SOP1.WORKER RESET PB SW
      AND     X53E  ; SAFETY AREA CUTAIN 1
      AND     X53F  ; SAFETY AREA CUTAIN 2
      OUT     M4811  ; SOP1.WORK.PB.START.RESERVE
377   LD      M4813  ; WORK.LOAD.PALLET.AUX
      AND     M4811  ; SOP1.WORK.PB.START.RESERVE
      AND     X53E  ; SAFETY AREA CUTAIN 1
      AND     X53F  ; SAFETY AREA CUTAIN 2
      OR      M4807  ; WORK.LOAD.PALLET.POSITION.DOWN
      AND     M4812  ; WORK.LOADING.2STEP.AUTO
      ANI     M4808  ; WORK.LOAD.STOPPER DOWN
      ANI     M4810  ; WORK.LOADING.AUTO.END
      OUT     M4807  ; WORK.LOAD.PALLET.POSITION.DOWN
      AND     X509  ; WORK LOADING PALLET POSI DN
      OUT     T4807 K5
391   LD      T4807
      AND     M4811  ; SOP1.WORK.PB.START.RESERVE
      ANI     M4820  ; REINLET.CONV.AUTO IN.CONV.MC.ON
      AND     X512  ; REINLET DIVERTER MID
      AND     X514  ; RE INLET DIVERTER PALLET DETECT
      OR      M4808  ; WORK.LOAD.STOPPER DOWN
      AND     M4812  ; WORK.LOADING.2STEP.AUTO
      ANI     M4809  ; WORK.LOAD.STOPPER UP
      OUT     M4808  ; WORK.LOAD.STOPPER DOWN
      ANI     X506  ; WORK LOADING STOPPER PALLET DETE
      OUT     T4808 K5
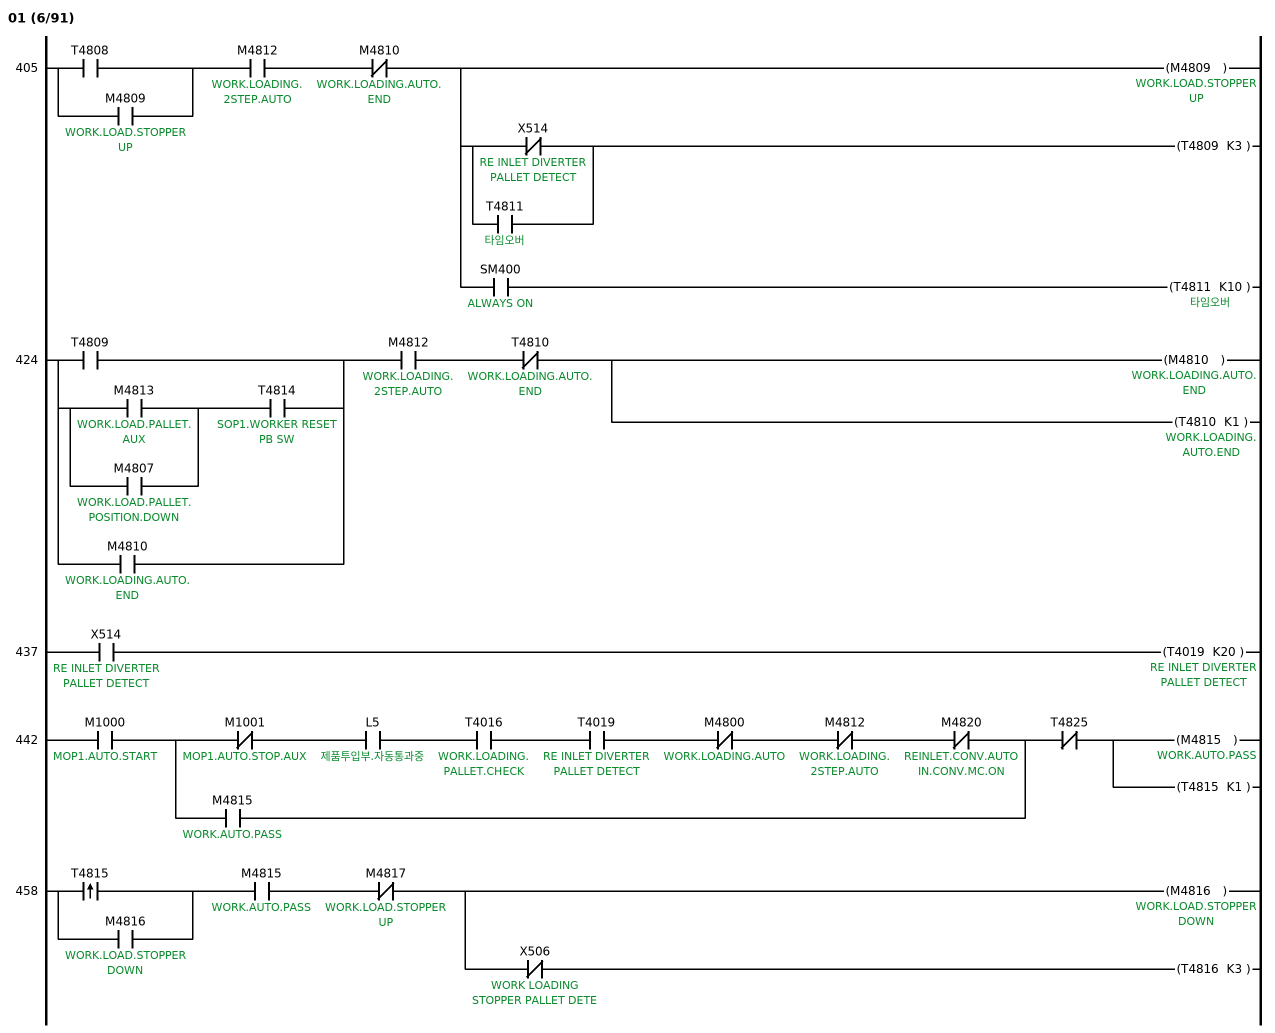
405   LD      T4808
      OR      M4809  ; WORK.LOAD.STOPPER UP
      AND     M4812  ; WORK.LOADING.2STEP.AUTO
      ANI     M4810  ; WORK.LOADING.AUTO.END
      OUT     M4809  ; WORK.LOAD.STOPPER UP
      MPS
      LDI     X514  ; RE INLET DIVERTER PALLET DETECT
      OR      T4811  ; 타임오버
      ANB
      OUT     T4809 K3
      MPP
      AND     SM400  ; ALWAYS ON
      OUT     T4811 K10  ; 타임오버
424   LD      T4809
      LD      M4813  ; WORK.LOAD.PALLET.AUX
      OR      M4807  ; WORK.LOAD.PALLET.POSITION.DOWN
      AND     T4814  ; SOP1.WORKER RESET PB SW
      ORB
      OR      M4810  ; WORK.LOADING.AUTO.END
      AND     M4812  ; WORK.LOADING.2STEP.AUTO
      ANI     T4810  ; WORK.LOADING.AUTO.END
      OUT     M4810  ; WORK.LOADING.AUTO.END
      OUT     T4810 K1  ; WORK.LOADING.AUTO.END
437   LD      X514  ; RE INLET DIVERTER PALLET DETECT
      OUT     T4019 K20  ; RE INLET DIVERTER PALLET DETECT
442   LD      M1000  ; MOP1.AUTO.START
      LDI     M1001  ; MOP1.AUTO.STOP.AUX
      AND     L5  ; 제품투입부.자동통과중
      AND     T4016  ; WORK.LOADING.PALLET.CHECK
      AND     T4019  ; RE INLET DIVERTER PALLET DETECT
      ANI     M4800  ; WORK.LOADING.AUTO
      ANI     M4812  ; WORK.LOADING.2STEP.AUTO
      ANI     M4820  ; REINLET.CONV.AUTO IN.CONV.MC.ON
      OR      M4815  ; WORK.AUTO.PASS
      ANB
      ANI     T4825
      OUT     M4815  ; WORK.AUTO.PASS
      OUT     T4815 K1
458   LDP     T4815
      OR      M4816  ; WORK.LOAD.STOPPER DOWN
      AND     M4815  ; WORK.AUTO.PASS
      ANI     M4817  ; WORK.LOAD.STOPPER UP
      OUT     M4816  ; WORK.LOAD.STOPPER DOWN
      ANI     X506  ; WORK LOADING STOPPER PALLET DETE
      OUT     T4816 K3
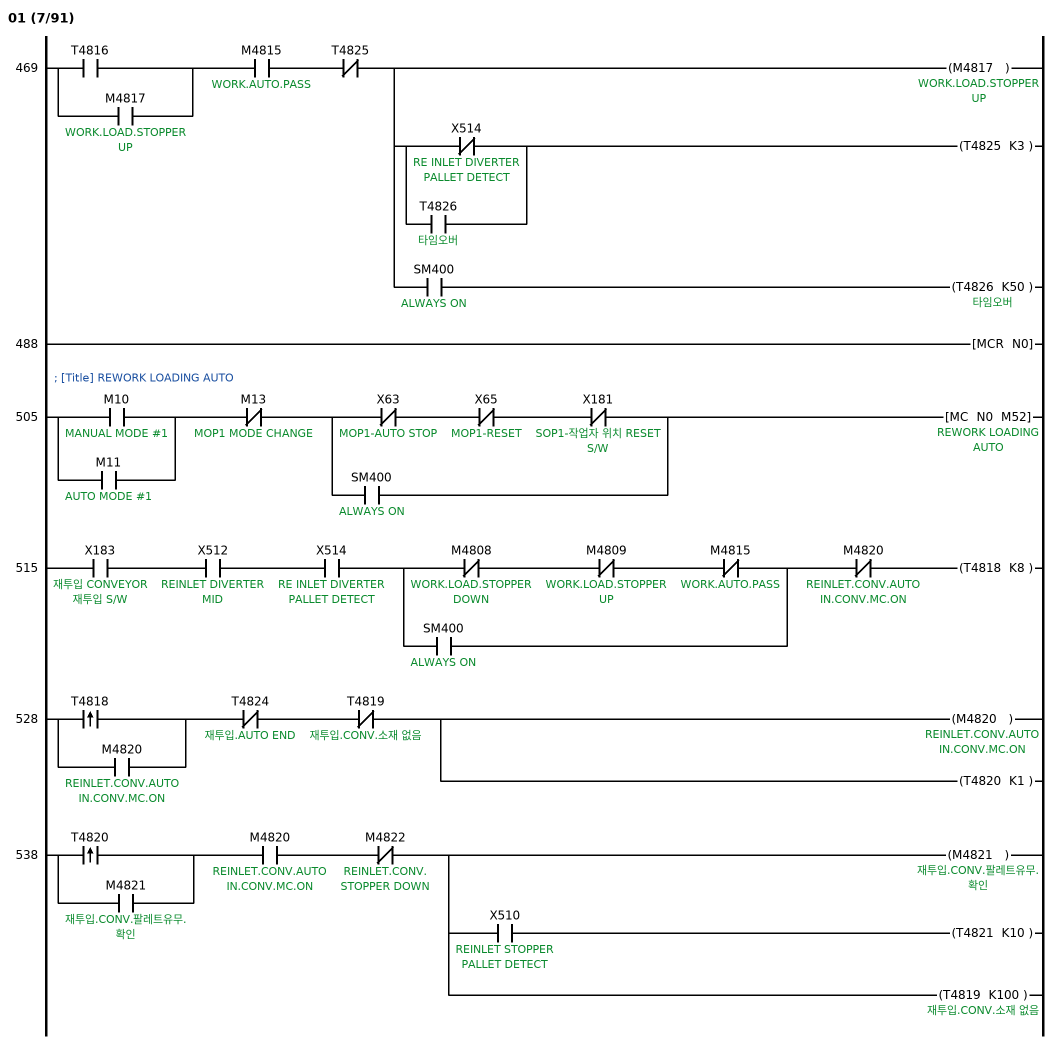
469   LD      T4816
      OR      M4817  ; WORK.LOAD.STOPPER UP
      AND     M4815  ; WORK.AUTO.PASS
      ANI     T4825
      OUT     M4817  ; WORK.LOAD.STOPPER UP
      MPS
      LDI     X514  ; RE INLET DIVERTER PALLET DETECT
      OR      T4826  ; 타임오버
      ANB
      OUT     T4825 K3
      MPP
      AND     SM400  ; ALWAYS ON
      OUT     T4826 K50  ; 타임오버
488   MCR     N0
; [Title] REWORK LOADING AUTO
505   LD      M10  ; MANUAL MODE #1
      OR      M11  ; AUTO MODE #1
      ANI     M13  ; MOP1 MODE CHANGE
      LDI     X63  ; MOP1-AUTO STOP
      ANI     X65  ; MOP1-RESET
      ANI     X181  ; SOP1-작업자 위치 RESET S/W
      OR      SM400  ; ALWAYS ON
      ANB
      MC      N0 M52  ; REWORK LOADING AUTO
515   LD      X183  ; 재투입 CONVEYOR 재투입 S/W
      AND     X512  ; REINLET DIVERTER MID
      AND     X514  ; RE INLET DIVERTER PALLET DETECT
      LDI     M4808  ; WORK.LOAD.STOPPER DOWN
      ANI     M4809  ; WORK.LOAD.STOPPER UP
      ANI     M4815  ; WORK.AUTO.PASS
      OR      SM400  ; ALWAYS ON
      ANB
      ANI     M4820  ; REINLET.CONV.AUTO IN.CONV.MC.ON
      OUT     T4818 K8
528   LDP     T4818
      OR      M4820  ; REINLET.CONV.AUTO IN.CONV.MC.ON
      ANI     T4824  ; 재투입.AUTO END
      ANI     T4819  ; 재투입.CONV.소재 없음
      OUT     M4820  ; REINLET.CONV.AUTO IN.CONV.MC.ON
      OUT     T4820 K1
538   LDP     T4820
      OR      M4821  ; 재투입.CONV.팔레트유무.확인
      AND     M4820  ; REINLET.CONV.AUTO IN.CONV.MC.ON
      ANI     M4822  ; REINLET.CONV.STOPPER DOWN
      OUT     M4821  ; 재투입.CONV.팔레트유무.확인
      MPS
      AND     X510  ; REINLET STOPPER PALLET DETECT
      OUT     T4821 K10
      MPP
      OUT     T4819 K100  ; 재투입.CONV.소재 없음
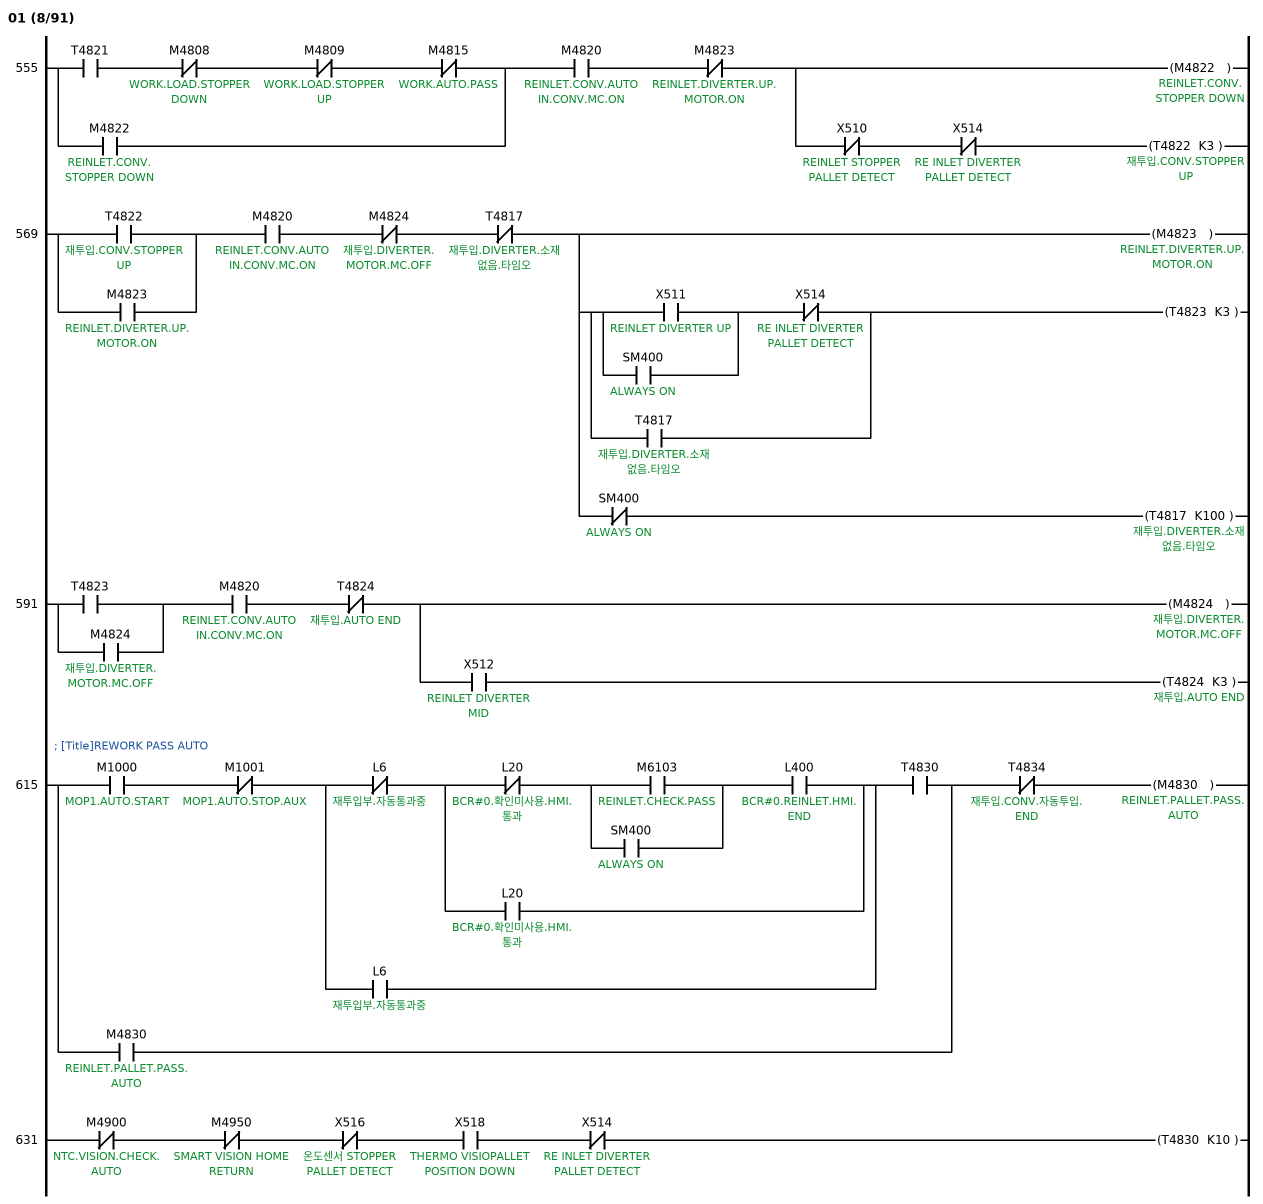
555   LD      T4821
      ANI     M4808  ; WORK.LOAD.STOPPER DOWN
      ANI     M4809  ; WORK.LOAD.STOPPER UP
      ANI     M4815  ; WORK.AUTO.PASS
      OR      M4822  ; REINLET.CONV.STOPPER DOWN
      AND     M4820  ; REINLET.CONV.AUTO IN.CONV.MC.ON
      ANI     M4823  ; REINLET.DIVERTER.UP.MOTOR.ON
      OUT     M4822  ; REINLET.CONV.STOPPER DOWN
      ANI     X510  ; REINLET STOPPER PALLET DETECT
      ANI     X514  ; RE INLET DIVERTER PALLET DETECT
      OUT     T4822 K3  ; 재투입.CONV.STOPPER UP
569   LD      T4822  ; 재투입.CONV.STOPPER UP
      OR      M4823  ; REINLET.DIVERTER.UP.MOTOR.ON
      AND     M4820  ; REINLET.CONV.AUTO IN.CONV.MC.ON
      ANI     M4824  ; 재투입.DIVERTER.MOTOR.MC.OFF
      ANI     T4817  ; 재투입.DIVERTER.소재 없음.타임오
      OUT     M4823  ; REINLET.DIVERTER.UP.MOTOR.ON
      MPS
      LD      X511  ; REINLET DIVERTER UP
      OR      SM400  ; ALWAYS ON
      ANI     X514  ; RE INLET DIVERTER PALLET DETECT
      OR      T4817  ; 재투입.DIVERTER.소재 없음.타임오
      ANB
      OUT     T4823 K3
      MPP
      ANI     SM400  ; ALWAYS ON
      OUT     T4817 K100  ; 재투입.DIVERTER.소재 없음.타임오
591   LD      T4823
      OR      M4824  ; 재투입.DIVERTER.MOTOR.MC.OFF
      AND     M4820  ; REINLET.CONV.AUTO IN.CONV.MC.ON
      ANI     T4824  ; 재투입.AUTO END
      OUT     M4824  ; 재투입.DIVERTER.MOTOR.MC.OFF
      AND     X512  ; REINLET DIVERTER MID
      OUT     T4824 K3  ; 재투입.AUTO END
; [Title]REWORK PASS AUTO
615   LD      M1000  ; MOP1.AUTO.START
      ANI     M1001  ; MOP1.AUTO.STOP.AUX
      LDI     L6  ; 재투입부.자동통과중
      LDI     L20  ; BCR#0.확인미사용.HMI.통과
      LD      M6103  ; REINLET.CHECK.PASS
      OR      SM400  ; ALWAYS ON
      ANB
      AND     L400  ; BCR#0.REINLET.HMI.END
      OR      L20  ; BCR#0.확인미사용.HMI.통과
      ANB
      OR      L6  ; 재투입부.자동통과중
      ANB
      AND     T4830
      OR      M4830  ; REINLET.PALLET.PASS.AUTO
      ANI     T4834  ; 재투입.CONV.자동투입.END
      OUT     M4830  ; REINLET.PALLET.PASS.AUTO
631   LDI     M4900  ; NTC.VISION.CHECK.AUTO
      ANI     M4950  ; SMART VISION HOME RETURN
      ANI     X516  ; 온도센서 STOPPER PALLET DETECT
      AND     X518  ; THERMO VISIOPALLET POSITION DOWN
      ANI     X514  ; RE INLET DIVERTER PALLET DETECT
      OUT     T4830 K10
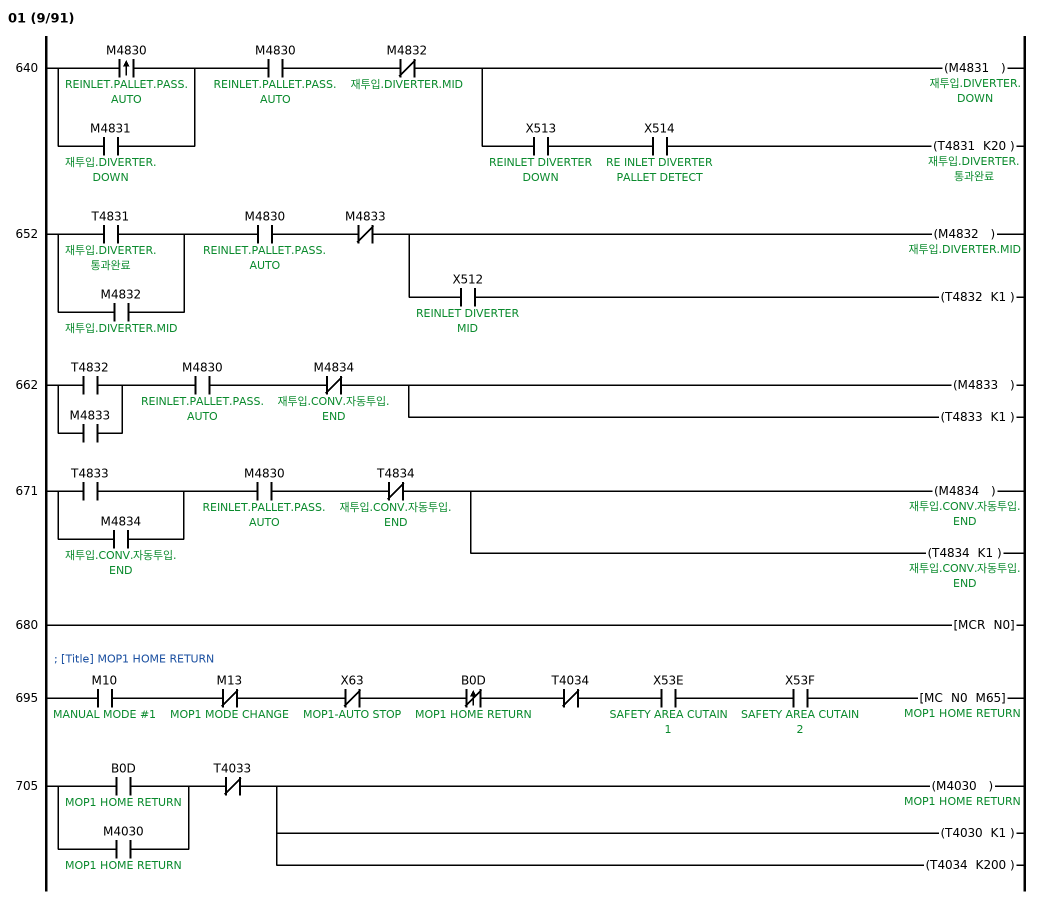
640   LDP     M4830  ; REINLET.PALLET.PASS.AUTO
      OR      M4831  ; 재투입.DIVERTER.DOWN
      AND     M4830  ; REINLET.PALLET.PASS.AUTO
      ANI     M4832  ; 재투입.DIVERTER.MID
      OUT     M4831  ; 재투입.DIVERTER.DOWN
      AND     X513  ; REINLET DIVERTER DOWN
      AND     X514  ; RE INLET DIVERTER PALLET DETECT
      OUT     T4831 K20  ; 재투입.DIVERTER.통과완료
652   LD      T4831  ; 재투입.DIVERTER.통과완료
      OR      M4832  ; 재투입.DIVERTER.MID
      AND     M4830  ; REINLET.PALLET.PASS.AUTO
      ANI     M4833
      OUT     M4832  ; 재투입.DIVERTER.MID
      AND     X512  ; REINLET DIVERTER MID
      OUT     T4832 K1
662   LD      T4832
      OR      M4833
      AND     M4830  ; REINLET.PALLET.PASS.AUTO
      ANI     M4834  ; 재투입.CONV.자동투입.END
      OUT     M4833
      OUT     T4833 K1
671   LD      T4833
      OR      M4834  ; 재투입.CONV.자동투입.END
      AND     M4830  ; REINLET.PALLET.PASS.AUTO
      ANI     T4834  ; 재투입.CONV.자동투입.END
      OUT     M4834  ; 재투입.CONV.자동투입.END
      OUT     T4834 K1  ; 재투입.CONV.자동투입.END
680   MCR     N0
; [Title] MOP1 HOME RETURN
695   LD      M10  ; MANUAL MODE #1
      ANI     M13  ; MOP1 MODE CHANGE
      ANI     X63  ; MOP1-AUTO STOP
      ANDPI   B0D  ; MOP1 HOME RETURN
      ANI     T4034
      AND     X53E  ; SAFETY AREA CUTAIN 1
      AND     X53F  ; SAFETY AREA CUTAIN 2
      MC      N0 M65  ; MOP1 HOME RETURN
705   LD      B0D  ; MOP1 HOME RETURN
      OR      M4030  ; MOP1 HOME RETURN
      ANI     T4033
      OUT     M4030  ; MOP1 HOME RETURN
      OUT     T4030 K1
      OUT     T4034 K200
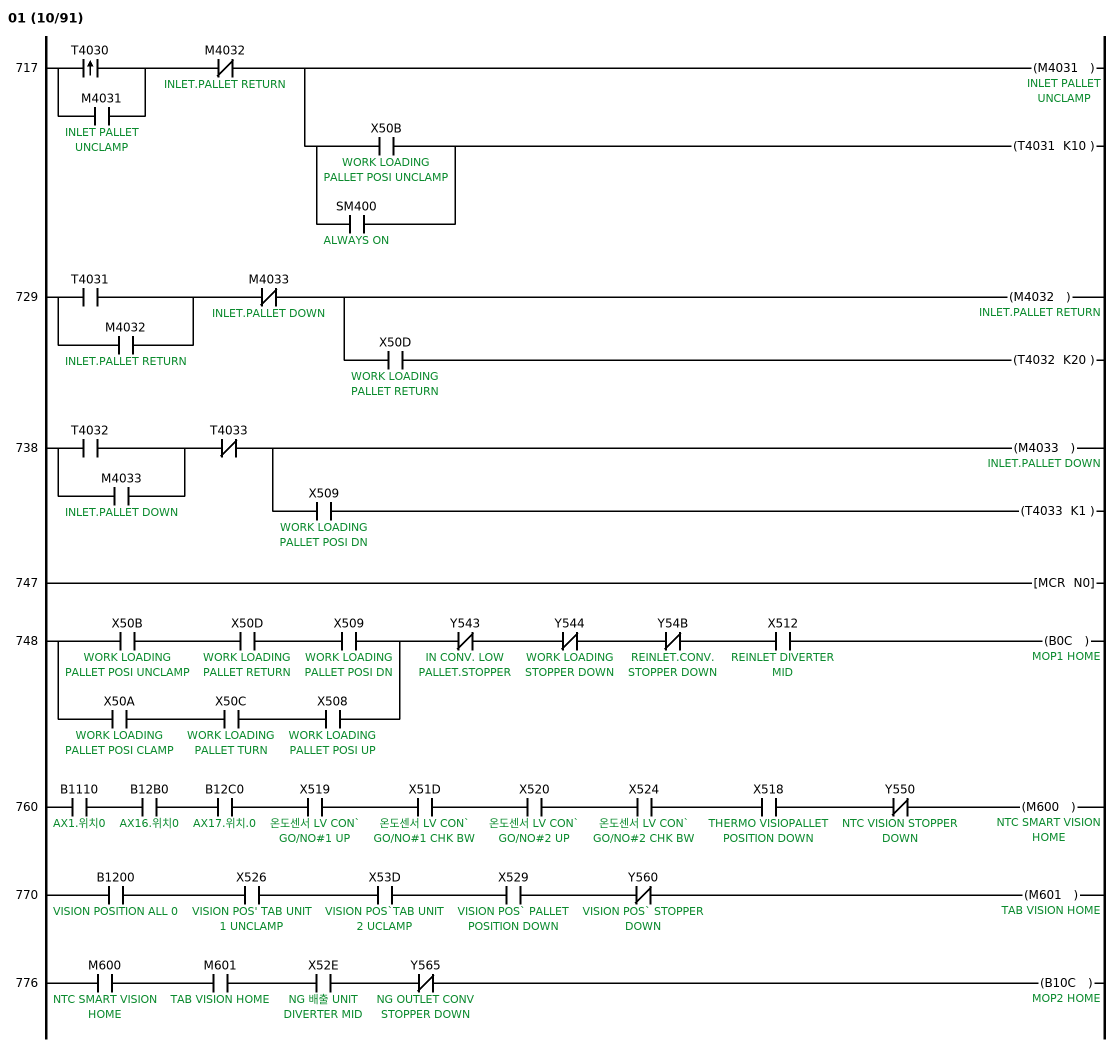
717   LDP     T4030
      OR      M4031  ; INLET PALLET UNCLAMP
      ANI     M4032  ; INLET.PALLET RETURN
      OUT     M4031  ; INLET PALLET UNCLAMP
      LD      X50B  ; WORK LOADING PALLET POSI UNCLAMP
      OR      SM400  ; ALWAYS ON
      ANB
      OUT     T4031 K10
729   LD      T4031
      OR      M4032  ; INLET.PALLET RETURN
      ANI     M4033  ; INLET.PALLET DOWN
      OUT     M4032  ; INLET.PALLET RETURN
      AND     X50D  ; WORK LOADING PALLET RETURN
      OUT     T4032 K20
738   LD      T4032
      OR      M4033  ; INLET.PALLET DOWN
      ANI     T4033
      OUT     M4033  ; INLET.PALLET DOWN
      AND     X509  ; WORK LOADING PALLET POSI DN
      OUT     T4033 K1
747   MCR     N0
748   LD      X50B  ; WORK LOADING PALLET POSI UNCLAMP
      AND     X50D  ; WORK LOADING PALLET RETURN
      AND     X509  ; WORK LOADING PALLET POSI DN
      LD      X50A  ; WORK LOADING PALLET POSI CLAMP
      AND     X50C  ; WORK LOADING PALLET TURN
      AND     X508  ; WORK LOADING PALLET POSI UP
      ORB
      ANI     Y543  ; IN CONV. LOW PALLET.STOPPER
      ANI     Y544  ; WORK LOADING STOPPER DOWN
      ANI     Y54B  ; REINLET.CONV.STOPPER DOWN
      AND     X512  ; REINLET DIVERTER MID
      OUT     B0C  ; MOP1 HOME
760   LD      B1110  ; AX1.위치0
      AND     B12B0  ; AX16.위치0
      AND     B12C0  ; AX17.위치.0
      AND     X519  ; 온도센서 LV CON` GO/NO#1 UP
      AND     X51D  ; 온도센서 LV CON` GO/NO#1 CHK BW
      AND     X520  ; 온도센서 LV CON` GO/NO#2 UP
      AND     X524  ; 온도센서 LV CON` GO/NO#2 CHK BW
      AND     X518  ; THERMO VISIOPALLET POSITION DOWN
      ANI     Y550  ; NTC VISION STOPPER DOWN
      OUT     M600  ; NTC SMART VISION HOME
770   LD      B1200  ; VISION POSITION ALL 0
      AND     X526  ; VISION POS' TAB UNIT 1 UNCLAMP
      AND     X53D  ; VISION POS`TAB UNIT 2 UCLAMP
      AND     X529  ; VISION POS` PALLET POSITION DOWN
      ANI     Y560  ; VISION POS` STOPPER DOWN
      OUT     M601  ; TAB VISION HOME
776   LD      M600  ; NTC SMART VISION HOME
      AND     M601  ; TAB VISION HOME
      AND     X52E  ; NG 배출 UNIT DIVERTER MID
      ANI     Y565  ; NG OUTLET CONV STOPPER DOWN
      OUT     B10C  ; MOP2 HOME
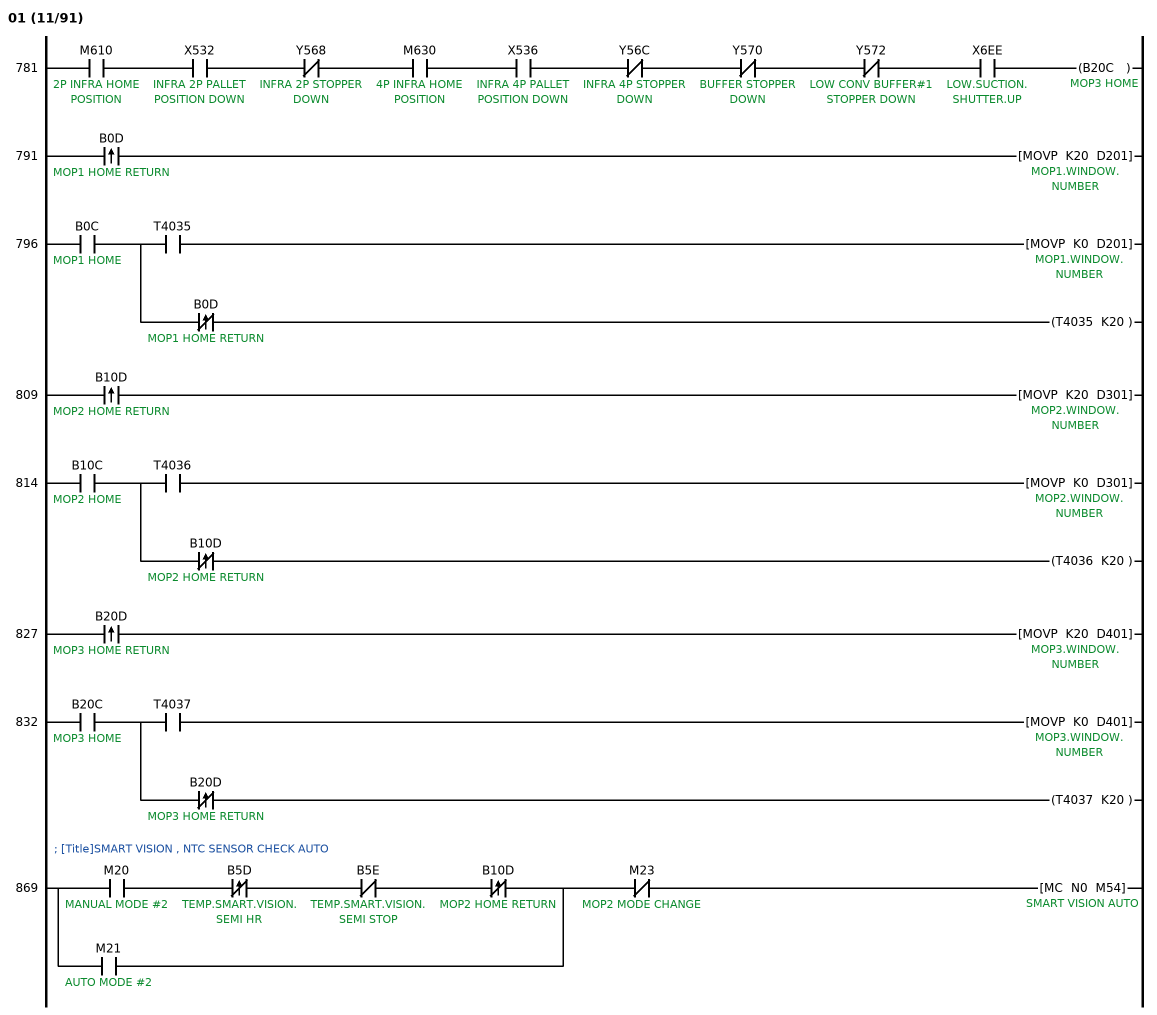
781   LD      M610  ; 2P INFRA HOME POSITION
      AND     X532  ; INFRA 2P PALLET POSITION DOWN
      ANI     Y568  ; INFRA 2P STOPPER DOWN
      AND     M630  ; 4P INFRA HOME POSITION
      AND     X536  ; INFRA 4P PALLET POSITION DOWN
      ANI     Y56C  ; INFRA 4P STOPPER DOWN
      ANI     Y570  ; BUFFER STOPPER DOWN
      ANI     Y572  ; LOW CONV BUFFER#1 STOPPER DOWN
      AND     X6EE  ; LOW.SUCTION.SHUTTER.UP
      OUT     B20C  ; MOP3 HOME
791   LDP     B0D  ; MOP1 HOME RETURN
      MOVP    K20 D201  ; MOP1.WINDOW.NUMBER
796   LD      B0C  ; MOP1 HOME
      MPS
      AND     T4035
      MOVP    K0 D201
      MPP
      ANDPI   B0D  ; MOP1 HOME RETURN
      OUT     T4035 K20
809   LDP     B10D  ; MOP2 HOME RETURN
      MOVP    K20 D301  ; MOP2.WINDOW.NUMBER
814   LD      B10C  ; MOP2 HOME
      MPS
      AND     T4036
      MOVP    K0 D301
      MPP
      ANDPI   B10D  ; MOP2 HOME RETURN
      OUT     T4036 K20
827   LDP     B20D  ; MOP3 HOME RETURN
      MOVP    K20 D401  ; MOP3.WINDOW.NUMBER
832   LD      B20C  ; MOP3 HOME
      MPS
      AND     T4037
      MOVP    K0 D401
      MPP
      ANDPI   B20D  ; MOP3 HOME RETURN
      OUT     T4037 K20
; [Title]SMART VISION , NTC SENSOR CHECK AUTO
869   LD      M20  ; MANUAL MODE #2
      ANDPI   B5D  ; TEMP.SMART.VISION.SEMI HR
      ANI     B5E  ; TEMP.SMART.VISION.SEMI STOP
      ANDPI   B10D  ; MOP2 HOME RETURN
      OR      M21  ; AUTO MODE #2
      ANI     M23  ; MOP2 MODE CHANGE
      MC      N0 M54  ; SMART VISION AUTO
